	UF : 7, UT : 3,	CONFIG : 'F U T, 0, 0, 0',
	X =   -66.816  mm,	Y =   342.344  mm,	Z =     0.000  mm,
	W =  -167.363 deg,	P =     0.000 deg,	R =  -154.099 deg
};
P[1214]{
   GP1:
	UF : 7, UT : 3,	CONFIG : 'F U T, 0, 0, 0',
	X =   -66.816  mm,	Y =   342.344  mm,	Z =     0.000  mm,
	W =  -167.363 deg,	P =     0.000 deg,	R =  -154.099 deg
};
P[1215]{
   GP1:
	UF : 7, UT : 3,	CONFIG : 'F U T, 0, 0, 0',
	X =   -66.816  mm,	Y =   342.344  mm,	Z =     0.000  mm,
	W =  -167.363 deg,	P =     0.000 deg,	R =  -154.099 deg
};
P[1216]{
   GP1:
	UF : 7, UT : 3,	CONFIG : 'F U T, 0, 0, 0',
	X =   -46.005  mm,	Y =   345.765  mm,	Z =     0.000  mm,
	W =  -167.363 deg,	P =     0.000 deg,	R =  -157.374 deg
};
P[1217]{
   GP1:
	UF : 7, UT : 3,	CONFIG : 'F U T, 0, 0, 0',
	X =   -26.635  mm,	Y =   347.781  mm,	Z =     0.000  mm,
	W =  -167.364 deg,	P =     0.000 deg,	R =  -160.858 deg
};
P[1218]{
   GP1:
	UF : 7, UT : 3,	CONFIG : 'F U T, 0, 0, 0',
	X =   -26.635  mm,	Y =   347.781  mm,	Z =     0.000  mm,
	W =  -167.364 deg,	P =     0.000 deg,	R =  -160.858 deg
};
P[1219]{
   GP1:
	UF : 7, UT : 3,	CONFIG : 'F U T, 0, 0, 0',
	X =   -26.635  mm,	Y =   347.781  mm,	Z =     0.000  mm,
	W =  -167.364 deg,	P =     0.000 deg,	R =  -160.858 deg
};
P[1220]{
   GP1:
	UF : 7, UT : 3,	CONFIG : 'F U T, 0, 0, 0',
	X =   -26.635  mm,	Y =   347.781  mm,	Z =     0.000  mm,
	W =  -167.364 deg,	P =     0.000 deg,	R =  -160.858 deg
};
P[1221]{
   GP1:
	UF : 7, UT : 3,	CONFIG : 'F U T, 0, 0, 0',
	X =    26.635  mm,	Y =   347.781  mm,	Z =     0.000  mm,
	W =  -167.363 deg,	P =     0.000 deg,	R =  -169.046 deg
};
P[1222]{
   GP1:
	UF : 7, UT : 3,	CONFIG : 'F U T, 0, 0, 0',
	X =    26.635  mm,	Y =   347.781  mm,	Z =     0.000  mm,
	W =  -167.363 deg,	P =     0.000 deg,	R =  -169.046 deg
};
P[1223]{
   GP1:
	UF : 7, UT : 3,	CONFIG : 'F U T, 0, 0, 0',
	X =    26.635  mm,	Y =   347.781  mm,	Z =     0.000  mm,
	W =  -167.363 deg,	P =     0.000 deg,	R =  -169.046 deg
};
P[1224]{
   GP1:
	UF : 7, UT : 3,	CONFIG : 'F U T, 0, 0, 0',
	X =    26.635  mm,	Y =   347.781  mm,	Z =     0.000  mm,
	W =  -167.363 deg,	P =     0.000 deg,	R =  -169.046 deg
};
P[1225]{
   GP1:
	UF : 7, UT : 3,	CONFIG : 'F U T, 0, 0, 0',
	X =    45.934  mm,	Y =   345.776  mm,	Z =     0.000  mm,
	W =  -167.363 deg,	P =     0.000 deg,	R =  -172.500 deg
};
P[1226]{
   GP1:
	UF : 7, UT : 3,	CONFIG : 'F U T, 0, 0, 0',
	X =    66.816  mm,	Y =   342.344  mm,	Z =     0.000  mm,
	W =  -167.363 deg,	P =     0.000 deg,	R =  -175.771 deg
};
P[1227]{
   GP1:
	UF : 7, UT : 3,	CONFIG : 'F U T, 0, 0, 0',
	X =    66.816  mm,	Y =   342.344  mm,	Z =     0.000  mm,
	W =  -167.363 deg,	P =     0.000 deg,	R =  -175.771 deg
};
P[1228]{
   GP1:
	UF : 7, UT : 3,	CONFIG : 'F U T, 0, 0, 0',
	X =    66.816  mm,	Y =   342.344  mm,	Z =     0.000  mm,
	W =  -167.363 deg,	P =     0.000 deg,	R =  -175.771 deg
};
P[1229]{
   GP1:
	UF : 7, UT : 3,	CONFIG : 'F U T, 0, 0, 0',
	X =    66.816  mm,	Y =   342.344  mm,	Z =     0.000  mm,
	W =  -167.363 deg,	P =     0.000 deg,	R =  -175.771 deg
};
P[1230]{
   GP1:
	UF : 7, UT : 3,	CONFIG : 'F U T, 0, 0, 0',
	X =    88.319  mm,	Y =   337.433  mm,	Z =     0.000  mm,
	W =  -167.363 deg,	P =     0.000 deg,	R =  -179.012 deg
};
P[1231]{
   GP1:
	UF : 7, UT : 3,	CONFIG : 'F U T, 0, 0, 0',
	X =    88.319  mm,	Y =   337.433  mm,	Z =     0.000  mm,
	W =  -167.363 deg,	P =     0.000 deg,	R =  -179.012 deg
};
P[1232]{
   GP1:
	UF : 7, UT : 3,	CONFIG : 'F U T, 0, 0, 0',
	X =    88.319  mm,	Y =   337.433  mm,	Z =     0.000  mm,
	W =  -167.363 deg,	P =     0.000 deg,	R =  -179.012 deg
};
P[1233]{
   GP1:
	UF : 7, UT : 3,	CONFIG : 'F U T, 0, 0, 0',
	X =    88.319  mm,	Y =   337.433  mm,	Z =     0.000  mm,
	W =  -167.363 deg,	P =     0.000 deg,	R =  -179.012 deg
};
P[1234]{
   GP1:
	UF : 7, UT : 3,	CONFIG : 'F U T, 0, 0, 0',
	X =   106.083  mm,	Y =   332.287  mm,	Z =     0.000  mm,
	W =  -167.364 deg,	P =     0.000 deg,	R =   177.374 deg
};
P[1235]{
   GP1:
	UF : 7, UT : 3,	CONFIG : 'F U T, 0, 0, 0',
	X =   126.912  mm,	Y =   324.901  mm,	Z =     0.000  mm,
	W =  -167.364 deg,	P =     0.000 deg,	R =   174.134 deg
};
P[1236]{
   GP1:
	UF : 7, UT : 3,	CONFIG : 'F U T, 0, 0, 0',
	X =   126.912  mm,	Y =   324.901  mm,	Z =     0.000  mm,
	W =  -167.364 deg,	P =     0.000 deg,	R =   174.134 deg
};
P[1237]{
   GP1:
	UF : 7, UT : 3,	CONFIG : 'F U T, 0, 0, 0',
	X =   126.912  mm,	Y =   324.901  mm,	Z =     0.000  mm,
	W =  -167.364 deg,	P =     0.000 deg,	R =   174.134 deg
};
P[1238]{
   GP1:
	UF : 7, UT : 3,	CONFIG : 'F U T, 0, 0, 0',
	X =   126.912  mm,	Y =   324.901  mm,	Z =     0.000  mm,
	W =  -167.364 deg,	P =     0.000 deg,	R =   174.134 deg
};
P[1239]{
   GP1:
	UF : 7, UT : 3,	CONFIG : 'F U T, 0, 0, 0',
	X =   174.892  mm,	Y =   301.790  mm,	Z =     0.000  mm,
	W =  -167.364 deg,	P =     0.001 deg,	R =   165.335 deg
};
P[1240]{
   GP1:
	UF : 7, UT : 3,	CONFIG : 'F U T, 0, 0, 0',
	X =   174.892  mm,	Y =   301.790  mm,	Z =     0.000  mm,
	W =  -167.364 deg,	P =     0.001 deg,	R =   165.335 deg
};
P[1241]{
   GP1:
	UF : 7, UT : 3,	CONFIG : 'F U T, 0, 0, 0',
	X =   174.892  mm,	Y =   301.790  mm,	Z =     0.000  mm,
	W =  -167.364 deg,	P =     0.001 deg,	R =   165.335 deg
};
P[1242]{
   GP1:
	UF : 7, UT : 3,	CONFIG : 'F U T, 0, 0, 0',
	X =   174.892  mm,	Y =   301.790  mm,	Z =     0.000  mm,
	W =  -167.364 deg,	P =     0.001 deg,	R =   165.335 deg
};
P[1243]{
   GP1:
	UF : 7, UT : 3,	CONFIG : 'F U T, 0, 0, 0',
	X =   191.564  mm,	Y =   291.498  mm,	Z =     0.000  mm,
	W =  -167.364 deg,	P =     0.000 deg,	R =   161.703 deg
};
P[1244]{
   GP1:
	UF : 7, UT : 3,	CONFIG : 'F U T, 0, 0, 0',
	X =   208.616  mm,	Y =   279.549  mm,	Z =     0.000  mm,
	W =  -167.364 deg,	P =     0.000 deg,	R =   158.339 deg
};
P[1245]{
   GP1:
	UF : 7, UT : 3,	CONFIG : 'F U T, 0, 0, 0',
	X =   224.914  mm,	Y =   266.601  mm,	Z =     0.001  mm,
	W =  -167.364 deg,	P =     0.000 deg,	R =   154.951 deg
};
P[1246]{
   GP1:
	UF : 7, UT : 3,	CONFIG : 'F U T, 0, 0, 0',
	X =   239.976  mm,	Y =   253.131  mm,	Z =     0.000  mm,
	W =  -167.365 deg,	P =     0.000 deg,	R =   151.474 deg
};
P[1247]{
   GP1:
	UF : 7, UT : 3,	CONFIG : 'F U T, 0, 0, 0',
	X =   255.318  mm,	Y =   237.661  mm,	Z =     0.000  mm,
	W =  -167.365 deg,	P =    -0.001 deg,	R =   148.214 deg
};
P[1248]{
   GP1:
	UF : 7, UT : 3,	CONFIG : 'F U T, 0, 0, 0',
	X =   255.318  mm,	Y =   237.661  mm,	Z =     0.000  mm,
	W =  -167.365 deg,	P =    -0.001 deg,	R =   148.214 deg
};
P[1249]{
   GP1:
	UF : 7, UT : 3,	CONFIG : 'F U T, 0, 0, 0',
	X =   255.318  mm,	Y =   237.661  mm,	Z =     0.000  mm,
	W =  -167.365 deg,	P =    -0.001 deg,	R =   148.214 deg
};
P[1250]{
   GP1:
	UF : 7, UT : 3,	CONFIG : 'F U T, 0, 0, 0',
	X =   255.318  mm,	Y =   237.661  mm,	Z =     0.000  mm,
	W =  -167.365 deg,	P =    -0.001 deg,	R =   148.214 deg
};
P[1251]{
   GP1:
	UF : 7, UT : 3,	CONFIG : 'F U T, 0, 0, 0',
	X =   288.517  mm,	Y =   196.042  mm,	Z =     0.000  mm,
	W =  -167.364 deg,	P =     0.001 deg,	R =   138.644 deg
};
P[1252]{
   GP1:
	UF : 7, UT : 3,	CONFIG : 'F U T, 0, 0, 0',
	X =   288.517  mm,	Y =   196.042  mm,	Z =     0.000  mm,
	W =  -167.364 deg,	P =     0.001 deg,	R =   138.644 deg
};
P[1253]{
   GP1:
	UF : 7, UT : 3,	CONFIG : 'F U T, 0, 0, 0',
	X =   288.517  mm,	Y =   196.042  mm,	Z =     0.000  mm,
	W =  -167.364 deg,	P =     0.001 deg,	R =   138.644 deg
};
P[1254]{
   GP1:
	UF : 7, UT : 3,	CONFIG : 'F U T, 0, 0, 0',
	X =   288.517  mm,	Y =   196.042  mm,	Z =     0.000  mm,
	W =  -167.364 deg,	P =     0.001 deg,	R =   138.644 deg
};
P[1255]{
   GP1:
	UF : 7, UT : 3,	CONFIG : 'F U T, 0, 0, 0',
	X =   300.602  mm,	Y =   176.942  mm,	Z =     0.000  mm,
	W =  -167.364 deg,	P =     0.000 deg,	R =   135.546 deg
};
P[1256]{
   GP1:
	UF : 7, UT : 3,	CONFIG : 'F U T, 0, 0, 0',
	X =   309.321  mm,	Y =   161.197  mm,	Z =     0.000  mm,
	W =  -167.363 deg,	P =     0.000 deg,	R =   132.101 deg
};
P[1257]{
   GP1:
	UF : 7, UT : 3,	CONFIG : 'F U T, 0, 0, 0',
	X =   309.321  mm,	Y =   161.197  mm,	Z =     0.000  mm,
	W =  -167.363 deg,	P =     0.000 deg,	R =   132.101 deg
};
P[1258]{
   GP1:
	UF : 7, UT : 3,	CONFIG : 'F U T, 0, 0, 0',
	X =   309.321  mm,	Y =   161.197  mm,	Z =     0.000  mm,
	W =  -167.363 deg,	P =     0.000 deg,	R =   132.101 deg
};
P[1259]{
   GP1:
	UF : 7, UT : 3,	CONFIG : 'F U T, 0, 0, 0',
	X =   309.321  mm,	Y =   161.197  mm,	Z =     0.000  mm,
	W =  -167.363 deg,	P =     0.000 deg,	R =   132.101 deg
};
P[1260]{
   GP1:
	UF : 7, UT : 3,	CONFIG : 'F U T, 0, 0, 0',
	X =   318.900  mm,	Y =   141.321  mm,	Z =     0.000  mm,
	W =  -167.363 deg,	P =     0.000 deg,	R =   128.500 deg
};
P[1261]{
   GP1:
	UF : 7, UT : 3,	CONFIG : 'F U T, 0, 0, 0',
	X =   318.900  mm,	Y =   141.321  mm,	Z =     0.000  mm,
	W =  -167.363 deg,	P =     0.000 deg,	R =   128.500 deg
};
P[1262]{
   GP1:
	UF : 7, UT : 3,	CONFIG : 'F U T, 0, 0, 0',
	X =   318.900  mm,	Y =   141.321  mm,	Z =     0.000  mm,
	W =  -167.363 deg,	P =     0.000 deg,	R =   128.500 deg
};
P[1263]{
   GP1:
	UF : 7, UT : 3,	CONFIG : 'F U T, 0, 0, 0',
	X =   318.900  mm,	Y =   141.321  mm,	Z =     0.000  mm,
	W =  -167.363 deg,	P =     0.000 deg,	R =   128.500 deg
};
P[1264]{
   GP1:
	UF : 7, UT : 3,	CONFIG : 'F U T, 0, 0, 0',
	X =   327.247  mm,	Y =   120.740  mm,	Z =     0.000  mm,
	W =  -167.364 deg,	P =     0.000 deg,	R =   125.297 deg
};
P[1265]{
   GP1:
	UF : 7, UT : 3,	CONFIG : 'F U T, 0, 0, 0',
	X =   333.135  mm,	Y =   103.355  mm,	Z =     0.000  mm,
	W =  -167.365 deg,	P =    -0.001 deg,	R =   121.761 deg
};
P[1266]{
   GP1:
	UF : 7, UT : 3,	CONFIG : 'F U T, 0, 0, 0',
	X =   333.135  mm,	Y =   103.355  mm,	Z =     0.000  mm,
	W =  -167.365 deg,	P =    -0.001 deg,	R =   121.761 deg
};
P[1267]{
   GP1:
	UF : 7, UT : 3,	CONFIG : 'F U T, 0, 0, 0',
	X =   333.135  mm,	Y =   103.355  mm,	Z =     0.000  mm,
	W =  -167.365 deg,	P =    -0.001 deg,	R =   121.761 deg
};
P[1268]{
   GP1:
	UF : 7, UT : 3,	CONFIG : 'F U T, 0, 0, 0',
	X =   333.135  mm,	Y =   103.355  mm,	Z =     0.000  mm,
	W =  -167.365 deg,	P =    -0.001 deg,	R =   121.761 deg
};
P[1269]{
   GP1:
	UF : 7, UT : 3,	CONFIG : 'F U T, 0, 0, 0',
	X =   344.991  mm,	Y =    51.425  mm,	Z =     0.000  mm,
	W =  -167.364 deg,	P =     0.001 deg,	R =   113.386 deg
};
P[1270]{
   GP1:
	UF : 7, UT : 3,	CONFIG : 'F U T, 0, 0, 0',
	X =   344.991  mm,	Y =    51.425  mm,	Z =     0.000  mm,
	W =  -167.364 deg,	P =     0.001 deg,	R =   113.386 deg
};
P[1271]{
   GP1:
	UF : 7, UT : 3,	CONFIG : 'F U T, 0, 0, 0',
	X =   344.991  mm,	Y =    51.425  mm,	Z =     0.000  mm,
	W =  -167.364 deg,	P =     0.001 deg,	R =   113.386 deg
};
P[1272]{
   GP1:
	UF : 7, UT : 3,	CONFIG : 'F U T, 0, 0, 0',
	X =   344.991  mm,	Y =    51.425  mm,	Z =     0.000  mm,
	W =  -167.364 deg,	P =     0.001 deg,	R =   113.386 deg
};
P[1273]{
   GP1:
	UF : 7, UT : 3,	CONFIG : 'F U T, 0, 0, 0',
	X =   347.736  mm,	Y =    27.239  mm,	Z =     0.000  mm,
	W =  -167.364 deg,	P =     0.000 deg,	R =   109.541 deg
};
P[1274]{
   GP1:
	UF : 7, UT : 3,	CONFIG : 'F U T, 0, 0, 0',
	X =   348.821  mm,	Y =     0.000  mm,	Z =     0.000  mm,
	W =  -167.364 deg,	P =    -0.001 deg,	R =   105.687 deg
};
P[1275]{
   GP1:
	UF : 7, UT : 3,	CONFIG : 'F U T, 0, 0, 0',
	X =   348.821  mm,	Y =     0.000  mm,	Z =     0.000  mm,
	W =  -167.364 deg,	P =    -0.001 deg,	R =   105.687 deg
};
P[1276]{
   GP1:
	UF : 7, UT : 3,	CONFIG : 'F U T, 0, 0, 0',
	X =   348.821  mm,	Y =     0.000  mm,	Z =     0.000  mm,
	W =  -167.364 deg,	P =    -0.001 deg,	R =   105.687 deg
};
P[1277]{
   GP1:
	UF : 7, UT : 3,	CONFIG : 'F U T, 0, 0, 0',
	X =   348.821  mm,	Y =     0.000  mm,	Z =     0.000  mm,
	W =  -167.364 deg,	P =    -0.001 deg,	R =   105.687 deg
};
P[1278]{
   GP1:
	UF : 7, UT : 3,	CONFIG : 'F U T, 0, 0, 0',
	X =   345.686  mm,	Y =     0.000  mm,	Z =     0.000  mm,
	W =  -167.364 deg,	P =    -0.001 deg,	R =   105.687 deg
};
P[1279]{
   GP1:
	UF : 7, UT : 3,	CONFIG : 'F U T, 0, 0, 0',
	X =   345.686  mm,	Y =     0.000  mm,	Z =     0.000  mm,
	W =  -167.364 deg,	P =    -0.001 deg,	R =   105.687 deg
};
P[1280]{
   GP1:
	UF : 7, UT : 3,	CONFIG : 'F U T, 0, 0, 0',
	X =   345.686  mm,	Y =     0.000  mm,	Z =     0.000  mm,
	W =  -167.364 deg,	P =    -0.001 deg,	R =   105.687 deg
};
P[1281]{
   GP1:
	UF : 7, UT : 3,	CONFIG : 'F U T, 0, 0, 0',
	X =   345.686  mm,	Y =     0.000  mm,	Z =     0.000  mm,
	W =  -167.364 deg,	P =    -0.001 deg,	R =   105.687 deg
};
P[1282]{
   GP1:
	UF : 7, UT : 3,	CONFIG : 'F U T, 0, 0, 0',
	X =   344.660  mm,	Y =    26.365  mm,	Z =     0.000  mm,
	W =  -167.364 deg,	P =     0.000 deg,	R =   109.418 deg
};
P[1283]{
   GP1:
	UF : 7, UT : 3,	CONFIG : 'F U T, 0, 0, 0',
	X =   342.332  mm,	Y =    47.913  mm,	Z =     0.000  mm,
	W =  -167.364 deg,	P =     0.001 deg,	R =   113.455 deg
};
P[1284]{
   GP1:
	UF : 7, UT : 3,	CONFIG : 'F U T, 0, 0, 0',
	X =   342.332  mm,	Y =    47.913  mm,	Z =     0.000  mm,
	W =  -167.364 deg,	P =     0.001 deg,	R =   113.455 deg
};
P[1285]{
   GP1:
	UF : 7, UT : 3,	CONFIG : 'F U T, 0, 0, 0',
	X =   342.332  mm,	Y =    47.913  mm,	Z =     0.000  mm,
	W =  -167.364 deg,	P =     0.001 deg,	R =   113.455 deg
};
P[1286]{
   GP1:
	UF : 7, UT : 3,	CONFIG : 'F U T, 0, 0, 0',
	X =   342.332  mm,	Y =    47.913  mm,	Z =     0.000  mm,
	W =  -167.364 deg,	P =     0.001 deg,	R =   113.455 deg
};
P[1287]{
   GP1:
	UF : 7, UT : 3,	CONFIG : 'F U T, 0, 0, 0',
	X =   329.241  mm,	Y =   105.355  mm,	Z =     0.000  mm,
	W =  -167.365 deg,	P =    -0.001 deg,	R =   123.426 deg
};
P[1288]{
   GP1:
	UF : 7, UT : 3,	CONFIG : 'F U T, 0, 0, 0',
	X =   329.241  mm,	Y =   105.355  mm,	Z =     0.000  mm,
	W =  -167.365 deg,	P =    -0.001 deg,	R =   123.426 deg
};
P[1289]{
   GP1:
	UF : 7, UT : 3,	CONFIG : 'F U T, 0, 0, 0',
	X =   329.241  mm,	Y =   105.355  mm,	Z =     0.000  mm,
	W =  -167.365 deg,	P =    -0.001 deg,	R =   123.426 deg
};
P[1290]{
   GP1:
	UF : 7, UT : 3,	CONFIG : 'F U T, 0, 0, 0',
	X =   329.241  mm,	Y =   105.355  mm,	Z =     0.000  mm,
	W =  -167.365 deg,	P =    -0.001 deg,	R =   123.426 deg
};
P[1291]{
   GP1:
	UF : 7, UT : 3,	CONFIG : 'F U T, 0, 0, 0',
	X =   321.435  mm,	Y =   127.175  mm,	Z =     0.000  mm,
	W =  -167.364 deg,	P =     0.000 deg,	R =   126.652 deg
};
P[1292]{
   GP1:
	UF : 7, UT : 3,	CONFIG : 'F U T, 0, 0, 0',
	X =   314.243  mm,	Y =   144.001  mm,	Z =     0.000  mm,
	W =  -167.363 deg,	P =     0.000 deg,	R =   130.454 deg
};
P[1293]{
   GP1:
	UF : 7, UT : 3,	CONFIG : 'F U T, 0, 0, 0',
	X =   314.243  mm,	Y =   144.001  mm,	Z =     0.000  mm,
	W =  -167.363 deg,	P =     0.000 deg,	R =   130.454 deg
};
P[1294]{
   GP1:
	UF : 7, UT : 3,	CONFIG : 'F U T, 0, 0, 0',
	X =   314.243  mm,	Y =   144.001  mm,	Z =     0.000  mm,
	W =  -167.363 deg,	P =     0.000 deg,	R =   130.454 deg
};
P[1295]{
   GP1:
	UF : 7, UT : 3,	CONFIG : 'F U T, 0, 0, 0',
	X =   314.243  mm,	Y =   144.001  mm,	Z =     0.000  mm,
	W =  -167.363 deg,	P =     0.000 deg,	R =   130.454 deg
};
P[1296]{
   GP1:
	UF : 7, UT : 3,	CONFIG : 'F U T, 0, 0, 0',
	X =   308.505  mm,	Y =   155.937  mm,	Z =     0.000  mm,
	W =  -167.363 deg,	P =     0.000 deg,	R =   132.305 deg
};
P[1297]{
   GP1:
	UF : 7, UT : 3,	CONFIG : 'F U T, 0, 0, 0',
	X =   308.505  mm,	Y =   155.937  mm,	Z =     0.000  mm,
	W =  -167.363 deg,	P =     0.000 deg,	R =   132.305 deg
};
P[1298]{
   GP1:
	UF : 7, UT : 3,	CONFIG : 'F U T, 0, 0, 0',
	X =   308.505  mm,	Y =   155.937  mm,	Z =     0.000  mm,
	W =  -167.363 deg,	P =     0.000 deg,	R =   132.305 deg
};
P[1299]{
   GP1:
	UF : 7, UT : 3,	CONFIG : 'F U T, 0, 0, 0',
	X =   308.505  mm,	Y =   155.937  mm,	Z =     0.000  mm,
	W =  -167.363 deg,	P =     0.000 deg,	R =   132.305 deg
};
P[1300]{
   GP1:
	UF : 7, UT : 3,	CONFIG : 'F U T, 0, 0, 0',
	X =   297.848  mm,	Y =   175.435  mm,	Z =     0.000  mm,
	W =  -167.364 deg,	P =     0.000 deg,	R =   135.574 deg
};
P[1301]{
   GP1:
	UF : 7, UT : 3,	CONFIG : 'F U T, 0, 0, 0',
	X =   287.641  mm,	Y =   191.697  mm,	Z =     0.000  mm,
	W =  -167.364 deg,	P =     0.001 deg,	R =   138.948 deg
};
P[1302]{
   GP1:
	UF : 7, UT : 3,	CONFIG : 'F U T, 0, 0, 0',
	X =   287.641  mm,	Y =   191.697  mm,	Z =     0.000  mm,
	W =  -167.364 deg,	P =     0.001 deg,	R =   138.948 deg
};
P[1303]{
   GP1:
	UF : 7, UT : 3,	CONFIG : 'F U T, 0, 0, 0',
	X =   287.641  mm,	Y =   191.697  mm,	Z =     0.000  mm,
	W =  -167.364 deg,	P =     0.001 deg,	R =   138.948 deg
};
P[1304]{
   GP1:
	UF : 7, UT : 3,	CONFIG : 'F U T, 0, 0, 0',
	X =   287.641  mm,	Y =   191.697  mm,	Z =     0.000  mm,
	W =  -167.364 deg,	P =     0.001 deg,	R =   138.948 deg
};
P[1305]{
   GP1:
	UF : 7, UT : 3,	CONFIG : 'F U T, 0, 0, 0',
	X =   250.901  mm,	Y =   237.773  mm,	Z =     0.000  mm,
	W =  -167.365 deg,	P =    -0.001 deg,	R =   148.657 deg
};
P[1306]{
   GP1:
	UF : 7, UT : 3,	CONFIG : 'F U T, 0, 0, 0',
	X =   250.901  mm,	Y =   237.773  mm,	Z =     0.000  mm,
	W =  -167.365 deg,	P =    -0.001 deg,	R =   148.657 deg
};
P[1307]{
   GP1:
	UF : 7, UT : 3,	CONFIG : 'F U T, 0, 0, 0',
	X =   250.901  mm,	Y =   237.773  mm,	Z =     0.000  mm,
	W =  -167.365 deg,	P =    -0.001 deg,	R =   148.657 deg
};
P[1308]{
   GP1:
	UF : 7, UT : 3,	CONFIG : 'F U T, 0, 0, 0',
	X =   250.901  mm,	Y =   237.773  mm,	Z =     0.000  mm,
	W =  -167.365 deg,	P =    -0.001 deg,	R =   148.657 deg
};
P[1309]{
   GP1:
	UF : 7, UT : 3,	CONFIG : 'F U T, 0, 0, 0',
	X =   233.996  mm,	Y =   254.423  mm,	Z =     0.000  mm,
	W =  -167.365 deg,	P =     0.000 deg,	R =   152.488 deg
};
P[1310]{
   GP1:
	UF : 7, UT : 3,	CONFIG : 'F U T, 0, 0, 0',
	X =   216.033  mm,	Y =   269.842  mm,	Z =     0.001  mm,
	W =  -167.364 deg,	P =     0.000 deg,	R =   156.343 deg
};
P[1311]{
   GP1:
	UF : 7, UT : 3,	CONFIG : 'F U T, 0, 0, 0',
	X =   197.478  mm,	Y =   283.704  mm,	Z =     0.000  mm,
	W =  -167.364 deg,	P =     0.000 deg,	R =   160.254 deg
};
P[1312]{
   GP1:
	UF : 7, UT : 3,	CONFIG : 'F U T, 0, 0, 0',
	X =   175.979  mm,	Y =   297.529  mm,	Z =     0.000  mm,
	W =  -167.364 deg,	P =     0.001 deg,	R =   164.017 deg
};
P[1313]{
   GP1:
	UF : 7, UT : 3,	CONFIG : 'F U T, 0, 0, 0',
	X =   175.979  mm,	Y =   297.529  mm,	Z =     0.000  mm,
	W =  -167.364 deg,	P =     0.001 deg,	R =   164.017 deg
};
P[1314]{
   GP1:
	UF : 7, UT : 3,	CONFIG : 'F U T, 0, 0, 0',
	X =   175.979  mm,	Y =   297.529  mm,	Z =     0.000  mm,
	W =  -167.364 deg,	P =     0.001 deg,	R =   164.017 deg
};
P[1315]{
   GP1:
	UF : 7, UT : 3,	CONFIG : 'F U T, 0, 0, 0',
	X =   175.979  mm,	Y =   297.529  mm,	Z =     0.000  mm,
	W =  -167.364 deg,	P =     0.001 deg,	R =   164.017 deg
};
P[1316]{
   GP1:
	UF : 7, UT : 3,	CONFIG : 'F U T, 0, 0, 0',
	X =   122.884  mm,	Y =   323.086  mm,	Z =     0.000  mm,
	W =  -167.364 deg,	P =     0.000 deg,	R =   173.711 deg
};
P[1317]{
   GP1:
	UF : 7, UT : 3,	CONFIG : 'F U T, 0, 0, 0',
	X =   122.884  mm,	Y =   323.086  mm,	Z =     0.000  mm,
	W =  -167.364 deg,	P =     0.000 deg,	R =   173.711 deg
};
P[1318]{
   GP1:
	UF : 7, UT : 3,	CONFIG : 'F U T, 0, 0, 0',
	X =   122.884  mm,	Y =   323.086  mm,	Z =     0.000  mm,
	W =  -167.364 deg,	P =     0.000 deg,	R =   173.711 deg
};
P[1319]{
   GP1:
	UF : 7, UT : 3,	CONFIG : 'F U T, 0, 0, 0',
	X =   122.884  mm,	Y =   323.086  mm,	Z =     0.000  mm,
	W =  -167.364 deg,	P =     0.000 deg,	R =   173.711 deg
};
P[1320]{
   GP1:
	UF : 7, UT : 3,	CONFIG : 'F U T, 0, 0, 0',
	X =   105.120  mm,	Y =   329.306  mm,	Z =     0.000  mm,
	W =  -167.364 deg,	P =     0.000 deg,	R =   177.352 deg
};
P[1321]{
   GP1:
	UF : 7, UT : 3,	CONFIG : 'F U T, 0, 0, 0',
	X =    83.393  mm,	Y =   335.476  mm,	Z =     0.000  mm,
	W =  -167.363 deg,	P =     0.000 deg,	R =  -179.548 deg
};
P[1322]{
   GP1:
	UF : 7, UT : 3,	CONFIG : 'F U T, 0, 0, 0',
	X =    83.393  mm,	Y =   335.476  mm,	Z =     0.000  mm,
	W =  -167.363 deg,	P =     0.000 deg,	R =  -179.548 deg
};
P[1323]{
   GP1:
	UF : 7, UT : 3,	CONFIG : 'F U T, 0, 0, 0',
	X =    83.393  mm,	Y =   335.476  mm,	Z =     0.000  mm,
	W =  -167.363 deg,	P =     0.000 deg,	R =  -179.548 deg
};
P[1324]{
   GP1:
	UF : 7, UT : 3,	CONFIG : 'F U T, 0, 0, 0',
	X =    83.393  mm,	Y =   335.476  mm,	Z =     0.000  mm,
	W =  -167.363 deg,	P =     0.000 deg,	R =  -179.548 deg
};
P[1325]{
   GP1:
	UF : 7, UT : 3,	CONFIG : 'F U T, 0, 0, 0',
	X =    70.462  mm,	Y =   338.412  mm,	Z =     0.000  mm,
	W =  -167.363 deg,	P =     0.000 deg,	R =  -177.098 deg
};
P[1326]{
   GP1:
	UF : 7, UT : 3,	CONFIG : 'F U T, 0, 0, 0',
	X =    70.462  mm,	Y =   338.412  mm,	Z =     0.000  mm,
	W =  -167.363 deg,	P =     0.000 deg,	R =  -177.098 deg
};
P[1327]{
   GP1:
	UF : 7, UT : 3,	CONFIG : 'F U T, 0, 0, 0',
	X =    70.462  mm,	Y =   338.412  mm,	Z =     0.000  mm,
	W =  -167.363 deg,	P =     0.000 deg,	R =  -177.098 deg
};
P[1328]{
   GP1:
	UF : 7, UT : 3,	CONFIG : 'F U T, 0, 0, 0',
	X =    70.462  mm,	Y =   338.412  mm,	Z =     0.000  mm,
	W =  -167.363 deg,	P =     0.000 deg,	R =  -177.098 deg
};
P[1329]{
   GP1:
	UF : 7, UT : 3,	CONFIG : 'F U T, 0, 0, 0',
	X =    51.004  mm,	Y =   341.888  mm,	Z =     0.000  mm,
	W =  -167.363 deg,	P =     0.000 deg,	R =  -173.340 deg
};
P[1330]{
   GP1:
	UF : 7, UT : 3,	CONFIG : 'F U T, 0, 0, 0',
	X =    29.459  mm,	Y =   344.419  mm,	Z =     0.000  mm,
	W =  -167.363 deg,	P =     0.000 deg,	R =  -169.941 deg
};
P[1331]{
   GP1:
	UF : 7, UT : 3,	CONFIG : 'F U T, 0, 0, 0',
	X =    29.459  mm,	Y =   344.419  mm,	Z =     0.000  mm,
	W =  -167.363 deg,	P =     0.000 deg,	R =  -169.941 deg
};
P[1332]{
   GP1:
	UF : 7, UT : 3,	CONFIG : 'F U T, 0, 0, 0',
	X =    29.459  mm,	Y =   344.419  mm,	Z =     0.000  mm,
	W =  -167.363 deg,	P =     0.000 deg,	R =  -169.941 deg
};
P[1333]{
   GP1:
	UF : 7, UT : 3,	CONFIG : 'F U T, 0, 0, 0',
	X =    29.459  mm,	Y =   344.419  mm,	Z =     0.000  mm,
	W =  -167.363 deg,	P =     0.000 deg,	R =  -169.941 deg
};
P[1334]{
   GP1:
	UF : 7, UT : 3,	CONFIG : 'F U T, 0, 0, 0',
	X =   -29.459  mm,	Y =   344.419  mm,	Z =     0.000  mm,
	W =  -167.364 deg,	P =     0.000 deg,	R =  -159.946 deg
};
P[1335]{
   GP1:
	UF : 7, UT : 3,	CONFIG : 'F U T, 0, 0, 0',
	X =   -29.459  mm,	Y =   344.419  mm,	Z =     0.000  mm,
	W =  -167.364 deg,	P =     0.000 deg,	R =  -159.946 deg
};
P[1336]{
   GP1:
	UF : 7, UT : 3,	CONFIG : 'F U T, 0, 0, 0',
	X =   -29.459  mm,	Y =   344.419  mm,	Z =     0.000  mm,
	W =  -167.364 deg,	P =     0.000 deg,	R =  -159.946 deg
};
P[1337]{
   GP1:
	UF : 7, UT : 3,	CONFIG : 'F U T, 0, 0, 0',
	X =   -29.459  mm,	Y =   344.419  mm,	Z =     0.000  mm,
	W =  -167.364 deg,	P =     0.000 deg,	R =  -159.946 deg
};
P[1338]{
   GP1:
	UF : 7, UT : 3,	CONFIG : 'F U T, 0, 0, 0',
	X =   -50.881  mm,	Y =   341.905  mm,	Z =     0.000  mm,
	W =  -167.363 deg,	P =     0.000 deg,	R =  -156.562 deg
};
P[1339]{
   GP1:
	UF : 7, UT : 3,	CONFIG : 'F U T, 0, 0, 0',
	X =   -70.462  mm,	Y =   338.412  mm,	Z =     0.000  mm,
	W =  -167.363 deg,	P =     0.000 deg,	R =  -152.846 deg
};
P[1340]{
   GP1:
	UF : 7, UT : 3,	CONFIG : 'F U T, 0, 0, 0',
	X =   -70.462  mm,	Y =   338.412  mm,	Z =     0.000  mm,
	W =  -167.363 deg,	P =     0.000 deg,	R =  -152.846 deg
};
P[1341]{
   GP1:
	UF : 7, UT : 3,	CONFIG : 'F U T, 0, 0, 0',
	X =   -70.462  mm,	Y =   338.412  mm,	Z =     0.000  mm,
	W =  -167.363 deg,	P =     0.000 deg,	R =  -152.846 deg
};
P[1342]{
   GP1:
	UF : 7, UT : 3,	CONFIG : 'F U T, 0, 0, 0',
	X =   -70.462  mm,	Y =   338.412  mm,	Z =     0.000  mm,
	W =  -167.363 deg,	P =     0.000 deg,	R =  -152.846 deg
};
P[1343]{
   GP1:
	UF : 7, UT : 3,	CONFIG : 'F U T, 0, 0, 0',
	X =   -83.393  mm,	Y =   335.476  mm,	Z =     0.000  mm,
	W =  -167.363 deg,	P =     0.000 deg,	R =  -150.369 deg
};
P[1344]{
   GP1:
	UF : 7, UT : 3,	CONFIG : 'F U T, 0, 0, 0',
	X =   -83.393  mm,	Y =   335.476  mm,	Z =     0.000  mm,
	W =  -167.363 deg,	P =     0.000 deg,	R =  -150.369 deg
};
P[1345]{
   GP1:
	UF : 7, UT : 3,	CONFIG : 'F U T, 0, 0, 0',
	X =   -83.393  mm,	Y =   335.476  mm,	Z =     0.000  mm,
	W =  -167.363 deg,	P =     0.000 deg,	R =  -150.369 deg
};
P[1346]{
   GP1:
	UF : 7, UT : 3,	CONFIG : 'F U T, 0, 0, 0',
	X =   -83.393  mm,	Y =   335.476  mm,	Z =     0.000  mm,
	W =  -167.363 deg,	P =     0.000 deg,	R =  -150.369 deg
};
P[1347]{
   GP1:
	UF : 7, UT : 3,	CONFIG : 'F U T, 0, 0, 0',
	X =  -105.618  mm,	Y =   329.150  mm,	Z =     0.000  mm,
	W =  -167.364 deg,	P =     0.001 deg,	R =  -147.148 deg
};
P[1348]{
   GP1:
	UF : 7, UT : 3,	CONFIG : 'F U T, 0, 0, 0',
	X =  -122.884  mm,	Y =   323.086  mm,	Z =     0.000  mm,
	W =  -167.364 deg,	P =     0.002 deg,	R =  -143.543 deg
};
P[1349]{
   GP1:
	UF : 7, UT : 3,	CONFIG : 'F U T, 0, 0, 0',
	X =  -122.884  mm,	Y =   323.086  mm,	Z =     0.000  mm,
	W =  -167.364 deg,	P =     0.002 deg,	R =  -143.543 deg
};
P[1350]{
   GP1:
	UF : 7, UT : 3,	CONFIG : 'F U T, 0, 0, 0',
	X =  -122.884  mm,	Y =   323.086  mm,	Z =     0.000  mm,
	W =  -167.364 deg,	P =     0.002 deg,	R =  -143.543 deg
};
P[1351]{
   GP1:
	UF : 7, UT : 3,	CONFIG : 'F U T, 0, 0, 0',
	X =  -122.884  mm,	Y =   323.086  mm,	Z =     0.000  mm,
	W =  -167.364 deg,	P =     0.002 deg,	R =  -143.543 deg
};
P[1352]{
   GP1:
	UF : 7, UT : 3,	CONFIG : 'F U T, 0, 0, 0',
	X =  -175.979  mm,	Y =   297.529  mm,	Z =     0.000  mm,
	W =  -167.373 deg,	P =    -0.006 deg,	R =  -133.905 deg
};
P[1353]{
   GP1:
	UF : 7, UT : 3,	CONFIG : 'F U T, 0, 0, 0',
	X =  -175.979  mm,	Y =   297.529  mm,	Z =     0.000  mm,
	W =  -167.373 deg,	P =    -0.006 deg,	R =  -133.905 deg
};
P[1354]{
   GP1:
	UF : 7, UT : 3,	CONFIG : 'F U T, 0, 0, 0',
	X =  -175.979  mm,	Y =   297.529  mm,	Z =     0.000  mm,
	W =  -167.373 deg,	P =    -0.006 deg,	R =  -133.905 deg
};
P[1355]{
   GP1:
	UF : 7, UT : 3,	CONFIG : 'F U T, 0, 0, 0',
	X =  -175.979  mm,	Y =   297.529  mm,	Z =     0.000  mm,
	W =  -167.373 deg,	P =    -0.006 deg,	R =  -133.905 deg
};
P[1356]{
   GP1:
	UF : 7, UT : 3,	CONFIG : 'F U T, 0, 0, 0',
	X =  -195.500  mm,	Y =   285.077  mm,	Z =     0.006  mm,
	W =  -167.372 deg,	P =    -0.005 deg,	R =  -130.444 deg
};
P[1357]{
   GP1:
	UF : 7, UT : 3,	CONFIG : 'F U T, 0, 0, 0',
	X =  -212.838  mm,	Y =   272.387  mm,	Z =     0.014  mm,
	W =  -167.372 deg,	P =    -0.004 deg,	R =  -126.946 deg
};
P[1358]{
   GP1:
	UF : 7, UT : 3,	CONFIG : 'F U T, 0, 0, 0',
	X =  -229.364  mm,	Y =   258.615  mm,	Z =     0.020  mm,
	W =  -167.371 deg,	P =    -0.003 deg,	R =  -123.454 deg
};
P[1359]{
   GP1:
	UF : 7, UT : 3,	CONFIG : 'F U T, 0, 0, 0',
	X =  -240.307  mm,	Y =   248.477  mm,	Z =     0.016  mm,
	W =  -167.396 deg,	P =     0.051 deg,	R =  -120.994 deg
};
P[1360]{
   GP1:
	UF : 7, UT : 3,	CONFIG : 'F U T, 0, 0, 0',
	X =  -250.901  mm,	Y =   237.773  mm,	Z =     0.000  mm,
	W =  -167.417 deg,	P =     0.107 deg,	R =  -118.546 deg
};
P[1361]{
   GP1:
	UF : 7, UT : 3,	CONFIG : 'F U T, 0, 0, 0',
	X =  -250.901  mm,	Y =   237.773  mm,	Z =     0.000  mm,
	W =  -167.417 deg,	P =     0.107 deg,	R =  -118.546 deg
};
P[1362]{
   GP1:
	UF : 7, UT : 3,	CONFIG : 'F U T, 0, 0, 0',
	X =  -250.901  mm,	Y =   237.773  mm,	Z =     0.000  mm,
	W =  -167.417 deg,	P =     0.107 deg,	R =  -118.546 deg
};
P[1363]{
   GP1:
	UF : 7, UT : 3,	CONFIG : 'F U T, 0, 0, 0',
	X =  -250.901  mm,	Y =   237.773  mm,	Z =     0.000  mm,
	W =  -167.417 deg,	P =     0.107 deg,	R =  -118.546 deg
};
P[1364]{
   GP1:
	UF : 7, UT : 3,	CONFIG : 'F U T, 0, 0, 0',
	X =  -287.641  mm,	Y =   191.697  mm,	Z =     0.000  mm,
	W =  -168.063 deg,	P =    -0.468 deg,	R =  -108.824 deg
};
P[1365]{
   GP1:
	UF : 7, UT : 3,	CONFIG : 'F U T, 0, 0, 0',
	X =  -287.641  mm,	Y =   191.697  mm,	Z =     0.000  mm,
	W =  -168.063 deg,	P =    -0.468 deg,	R =  -108.824 deg
};
P[1366]{
   GP1:
	UF : 7, UT : 3,	CONFIG : 'F U T, 0, 0, 0',
	X =  -287.641  mm,	Y =   191.697  mm,	Z =     0.000  mm,
	W =  -168.063 deg,	P =    -0.468 deg,	R =  -108.824 deg
};
P[1367]{
   GP1:
	UF : 7, UT : 3,	CONFIG : 'F U T, 0, 0, 0',
	X =  -287.641  mm,	Y =   191.697  mm,	Z =     0.000  mm,
	W =  -168.063 deg,	P =    -0.468 deg,	R =  -108.824 deg
};
P[1368]{
   GP1:
	UF : 7, UT : 3,	CONFIG : 'F U T, 0, 0, 0',
	X =  -295.473  mm,	Y =   179.397  mm,	Z =     0.299  mm,
	W =  -168.371 deg,	P =    -1.524 deg,	R =  -106.124 deg
};
P[1369]{
   GP1:
	UF : 7, UT : 3,	CONFIG : 'F U T, 0, 0, 0',
	X =  -299.979  mm,	Y =   171.757  mm,	Z =     0.593  mm,
	W =  -168.582 deg,	P =    -1.678 deg,	R =  -104.715 deg
};
P[1370]{
   GP1:
	UF : 7, UT : 3,	CONFIG : 'F U T, 0, 0, 0',
	X =  -304.573  mm,	Y =   163.495  mm,	Z =     0.880  mm,
	W =  -168.711 deg,	P =    -1.083 deg,	R =  -103.238 deg
};
P[1371]{
   GP1:
	UF : 7, UT : 3,	CONFIG : 'F U T, 0, 0, 0',
	X =  -307.581  mm,	Y =   157.753  mm,	Z =     1.000  mm,
	W =  -168.635 deg,	P =    -0.392 deg,	R =  -101.948 deg
};
P[1372]{
   GP1:
	UF : 7, UT : 3,	CONFIG : 'F U T, 0, 0, 0',
	X =  -307.581  mm,	Y =   157.753  mm,	Z =     1.000  mm,
	W =  -168.635 deg,	P =    -0.392 deg,	R =  -101.948 deg
};
P[1373]{
   GP1:
	UF : 7, UT : 3,	CONFIG : 'F U T, 0, 0, 0',
	X =  -307.581  mm,	Y =   157.753  mm,	Z =     1.000  mm,
	W =  -168.635 deg,	P =    -0.392 deg,	R =  -101.948 deg
};
P[1374]{
   GP1:
	UF : 7, UT : 3,	CONFIG : 'F U T, 0, 0, 0',
	X =  -307.581  mm,	Y =   157.753  mm,	Z =     1.000  mm,
	W =  -168.635 deg,	P =    -0.392 deg,	R =  -101.948 deg
};
P[1375]{
   GP1:
	UF : 7, UT : 3,	CONFIG : 'F U T, 0, 0, 0',
	X =  -315.125  mm,	Y =   142.110  mm,	Z =     1.000  mm,
	W =  -168.019 deg,	P =     0.716 deg,	R =   -99.203 deg
};
P[1376]{
   GP1:
	UF : 7, UT : 3,	CONFIG : 'F U T, 0, 0, 0',
	X =  -315.125  mm,	Y =   142.110  mm,	Z =     1.000  mm,
	W =  -168.019 deg,	P =     0.716 deg,	R =   -99.203 deg
};
P[1377]{
   GP1:
	UF : 7, UT : 3,	CONFIG : 'F U T, 0, 0, 0',
	X =  -315.125  mm,	Y =   142.110  mm,	Z =     1.000  mm,
	W =  -168.019 deg,	P =     0.716 deg,	R =   -99.203 deg
};
P[1378]{
   GP1:
	UF : 7, UT : 3,	CONFIG : 'F U T, 0, 0, 0',
	X =  -315.125  mm,	Y =   142.110  mm,	Z =     1.000  mm,
	W =  -168.019 deg,	P =     0.716 deg,	R =   -99.203 deg
};
P[1379]{
   GP1:
	UF : 7, UT : 3,	CONFIG : 'F U T, 0, 0, 0',
	X =  -319.199  mm,	Y =   132.690  mm,	Z =     0.839  mm,
	W =  -167.800 deg,	P =     1.582 deg,	R =   -97.400 deg
};
P[1380]{
   GP1:
	UF : 7, UT : 3,	CONFIG : 'F U T, 0, 0, 0',
	X =  -322.114  mm,	Y =   125.444  mm,	Z =     0.586  mm,
	W =  -167.715 deg,	P =     2.330 deg,	R =   -96.138 deg
};
P[1381]{
   GP1:
	UF : 7, UT : 3,	CONFIG : 'F U T, 0, 0, 0',
	X =  -324.359  mm,	Y =   119.513  mm,	Z =     0.341  mm,
	W =  -167.697 deg,	P =     2.244 deg,	R =   -95.130 deg
};
P[1382]{
   GP1:
	UF : 7, UT : 3,	CONFIG : 'F U T, 0, 0, 0',
	X =  -329.241  mm,	Y =   105.355  mm,	Z =     0.000  mm,
	W =  -167.650 deg,	P =     0.556 deg,	R =   -93.318 deg
};
P[1383]{
   GP1:
	UF : 7, UT : 3,	CONFIG : 'F U T, 0, 0, 0',
	X =  -329.241  mm,	Y =   105.355  mm,	Z =     0.000  mm,
	W =  -167.650 deg,	P =     0.556 deg,	R =   -93.318 deg
};
P[1384]{
   GP1:
	UF : 7, UT : 3,	CONFIG : 'F U T, 0, 0, 0',
	X =  -329.241  mm,	Y =   105.355  mm,	Z =     0.000  mm,
	W =  -167.650 deg,	P =     0.556 deg,	R =   -93.318 deg
};
P[1385]{
   GP1:
	UF : 7, UT : 3,	CONFIG : 'F U T, 0, 0, 0',
	X =  -329.241  mm,	Y =   105.355  mm,	Z =     0.000  mm,
	W =  -167.650 deg,	P =     0.556 deg,	R =   -93.318 deg
};
P[1386]{
   GP1:
	UF : 7, UT : 3,	CONFIG : 'F U T, 0, 1, 0',
	X =  -342.332  mm,	Y =    47.913  mm,	Z =     0.000  mm,
	W =  -167.380 deg,	P =    -0.011 deg,	R =   -83.337 deg
};
P[1387]{
   GP1:
	UF : 7, UT : 3,	CONFIG : 'F U T, 0, 1, 0',
	X =  -342.332  mm,	Y =    47.913  mm,	Z =     0.000  mm,
	W =  -167.380 deg,	P =    -0.011 deg,	R =   -83.337 deg
};
P[1388]{
   GP1:
	UF : 7, UT : 3,	CONFIG : 'F U T, 0, 1, 0',
	X =  -342.332  mm,	Y =    47.913  mm,	Z =     0.000  mm,
	W =  -167.380 deg,	P =    -0.011 deg,	R =   -83.337 deg
};
P[1389]{
   GP1:
	UF : 7, UT : 3,	CONFIG : 'F U T, 0, 1, 0',
	X =  -342.332  mm,	Y =    47.913  mm,	Z =     0.000  mm,
	W =  -167.380 deg,	P =    -0.011 deg,	R =   -83.337 deg
};
P[1390]{
   GP1:
	UF : 7, UT : 3,	CONFIG : 'F U T, 0, 1, 0',
	X =  -344.705  mm,	Y =    25.816  mm,	Z =     0.003  mm,
	W =  -167.372 deg,	P =    -0.002 deg,	R =   -79.244 deg
};
P[1391]{
   GP1:
	UF : 7, UT : 3,	CONFIG : 'F U T, 0, 1, 0',
	X =  -345.686  mm,	Y =     0.000  mm,	Z =     0.000  mm,
	W =  -167.361 deg,	P =     0.008 deg,	R =   -75.603 deg
};
P[1392]{
   GP1:
	UF : 7, UT : 3,	CONFIG : 'F U T, 0, 1, 0',
	X =  -345.686  mm,	Y =     0.000  mm,	Z =     0.000  mm,
	W =  -167.361 deg,	P =     0.008 deg,	R =   -75.603 deg
};
P[1393]{
   GP1:
	UF : 7, UT : 3,	CONFIG : 'F U T, 0, 1, 0',
	X =  -345.686  mm,	Y =     0.000  mm,	Z =     0.000  mm,
	W =  -167.361 deg,	P =     0.008 deg,	R =   -75.603 deg
};
P[1394]{
   GP1:
	UF : 7, UT : 3,	CONFIG : 'F U T, 0, 1, 0',
	X =  -345.686  mm,	Y =     0.000  mm,	Z =     0.000  mm,
	W =  -167.361 deg,	P =     0.008 deg,	R =   -75.603 deg
};
P[1395]{
   GP1:
	UF : 7, UT : 3,	CONFIG : 'F U T, 0, 1, 0',
	X =  -342.552  mm,	Y =     0.000  mm,	Z =     0.000  mm,
	W =  -167.361 deg,	P =     0.008 deg,	R =   -75.584 deg
};
P[1396]{
   GP1:
	UF : 7, UT : 3,	CONFIG : 'F U T, 0, 1, 0',
	X =  -342.552  mm,	Y =     0.000  mm,	Z =     0.000  mm,
	W =  -167.361 deg,	P =     0.008 deg,	R =   -75.584 deg
};
P[1397]{
   GP1:
	UF : 7, UT : 3,	CONFIG : 'F U T, 0, 1, 0',
	X =  -342.552  mm,	Y =     0.000  mm,	Z =     0.000  mm,
	W =  -167.361 deg,	P =     0.008 deg,	R =   -75.584 deg
};
P[1398]{
   GP1:
	UF : 7, UT : 3,	CONFIG : 'F U T, 0, 1, 0',
	X =  -342.552  mm,	Y =     0.000  mm,	Z =     0.000  mm,
	W =  -167.361 deg,	P =     0.008 deg,	R =   -75.584 deg
};
P[1399]{
   GP1:
	UF : 7, UT : 3,	CONFIG : 'F U T, 0, 1, 0',
	X =  -341.800  mm,	Y =    22.656  mm,	Z =     0.002  mm,
	W =  -167.370 deg,	P =    -0.001 deg,	R =   -78.735 deg
};
P[1400]{
   GP1:
	UF : 7, UT : 3,	CONFIG : 'F U T, 0, 1, 0',
	X =  -339.575  mm,	Y =    45.037  mm,	Z =     0.000  mm,
	W =  -167.378 deg,	P =    -0.011 deg,	R =   -81.919 deg
};
P[1401]{
   GP1:
	UF : 7, UT : 3,	CONFIG : 'F U T, 0, 1, 0',
	X =  -339.575  mm,	Y =    45.037  mm,	Z =     0.000  mm,
	W =  -167.378 deg,	P =    -0.011 deg,	R =   -81.919 deg
};
P[1402]{
   GP1:
	UF : 7, UT : 3,	CONFIG : 'F U T, 0, 1, 0',
	X =  -339.575  mm,	Y =    45.037  mm,	Z =     0.000  mm,
	W =  -167.378 deg,	P =    -0.011 deg,	R =   -81.919 deg
};
P[1403]{
   GP1:
	UF : 7, UT : 3,	CONFIG : 'F U T, 0, 1, 0',
	X =  -339.575  mm,	Y =    45.037  mm,	Z =     0.000  mm,
	W =  -167.378 deg,	P =    -0.011 deg,	R =   -81.919 deg
};
P[1404]{
   GP1:
	UF : 7, UT : 3,	CONFIG : 'F U T, 0, 0, 0',
	X =  -325.470  mm,	Y =   106.765  mm,	Z =     0.000  mm,
	W =  -167.618 deg,	P =     0.684 deg,	R =   -93.130 deg
};
P[1405]{
   GP1:
	UF : 7, UT : 3,	CONFIG : 'F U T, 0, 0, 0',
	X =  -325.470  mm,	Y =   106.765  mm,	Z =     0.000  mm,
	W =  -167.618 deg,	P =     0.684 deg,	R =   -93.130 deg
};
P[1406]{
   GP1:
	UF : 7, UT : 3,	CONFIG : 'F U T, 0, 0, 0',
	X =  -325.470  mm,	Y =   106.765  mm,	Z =     0.000  mm,
	W =  -167.618 deg,	P =     0.684 deg,	R =   -93.130 deg
};
P[1407]{
   GP1:
	UF : 7, UT : 3,	CONFIG : 'F U T, 0, 0, 0',
	X =  -325.470  mm,	Y =   106.765  mm,	Z =     0.000  mm,
	W =  -167.618 deg,	P =     0.684 deg,	R =   -93.130 deg
};
P[1408]{
   GP1:
	UF : 7, UT : 3,	CONFIG : 'F U T, 0, 0, 0',
	X =  -321.597  mm,	Y =   117.970  mm,	Z =     0.274  mm,
	W =  -167.697 deg,	P =     2.153 deg,	R =   -95.041 deg
};
P[1409]{
   GP1:
	UF : 7, UT : 3,	CONFIG : 'F U T, 0, 0, 0',
	X =  -320.331  mm,	Y =   121.319  mm,	Z =     0.406  mm,
	W =  -167.738 deg,	P =     2.368 deg,	R =   -95.784 deg
};
P[1410]{
   GP1:
	UF : 7, UT : 3,	CONFIG : 'F U T, 0, 0, 0',
	X =  -319.155  mm,	Y =   124.393  mm,	Z =     0.534  mm,
	W =  -167.774 deg,	P =     2.363 deg,	R =   -96.124 deg
};
P[1411]{
   GP1:
	UF : 7, UT : 3,	CONFIG : 'F U T, 0, 0, 0',
	X =  -317.879  mm,	Y =   127.633  mm,	Z =     0.663  mm,
	W =  -167.841 deg,	P =     2.145 deg,	R =   -96.813 deg
};
P[1412]{
   GP1:
	UF : 7, UT : 3,	CONFIG : 'F U T, 0, 0, 0',
	X =  -313.909  mm,	Y =   137.100  mm,	Z =     0.908  mm,
	W =  -168.040 deg,	P =     1.025 deg,	R =   -98.473 deg
};
P[1413]{
   GP1:
	UF : 7, UT : 3,	CONFIG : 'F U T, 0, 0, 0',
	X =  -307.714  mm,	Y =   150.492  mm,	Z =     0.986  mm,
	W =  -168.440 deg,	P =     0.127 deg,	R =  -100.987 deg
};
P[1414]{
   GP1:
	UF : 7, UT : 3,	CONFIG : 'F U T, 0, 0, 0',
	X =  -301.389  mm,	Y =   162.785  mm,	Z =     0.801  mm,
	W =  -168.743 deg,	P =    -1.086 deg,	R =  -103.380 deg
};
P[1415]{
   GP1:
	UF : 7, UT : 3,	CONFIG : 'F U T, 0, 0, 0',
	X =  -298.728  mm,	Y =   167.639  mm,	Z =     0.646  mm,
	W =  -168.684 deg,	P =    -1.479 deg,	R =  -104.289 deg
};
P[1416]{
   GP1:
	UF : 7, UT : 3,	CONFIG : 'F U T, 0, 0, 0',
	X =  -293.943  mm,	Y =   175.865  mm,	Z =     0.335  mm,
	W =  -168.467 deg,	P =    -1.585 deg,	R =  -105.877 deg
};
P[1417]{
   GP1:
	UF : 7, UT : 3,	CONFIG : 'F U T, 0, 0, 0',
	X =  -286.401  mm,	Y =   187.899  mm,	Z =     0.000  mm,
	W =  -168.114 deg,	P =    -0.620 deg,	R =  -108.438 deg
};
P[1418]{
   GP1:
	UF : 7, UT : 3,	CONFIG : 'F U T, 0, 0, 0',
	X =  -286.401  mm,	Y =   187.899  mm,	Z =     0.000  mm,
	W =  -168.114 deg,	P =    -0.620 deg,	R =  -108.438 deg
};
P[1419]{
   GP1:
	UF : 7, UT : 3,	CONFIG : 'F U T, 0, 0, 0',
	X =  -286.401  mm,	Y =   187.899  mm,	Z =     0.000  mm,
	W =  -168.114 deg,	P =    -0.620 deg,	R =  -108.438 deg
};
P[1420]{
   GP1:
	UF : 7, UT : 3,	CONFIG : 'F U T, 0, 0, 0',
	X =  -286.401  mm,	Y =   187.899  mm,	Z =     0.000  mm,
	W =  -168.114 deg,	P =    -0.620 deg,	R =  -108.438 deg
};
P[1421]{
   GP1:
	UF : 7, UT : 3,	CONFIG : 'F U T, 0, 0, 0',
	X =  -246.913  mm,	Y =   237.408  mm,	Z =     0.000  mm,
	W =  -167.403 deg,	P =     0.109 deg,	R =  -118.143 deg
};
P[1422]{
   GP1:
	UF : 7, UT : 3,	CONFIG : 'F U T, 0, 0, 0',
	X =  -246.913  mm,	Y =   237.408  mm,	Z =     0.000  mm,
	W =  -167.403 deg,	P =     0.109 deg,	R =  -118.143 deg
};
P[1423]{
   GP1:
	UF : 7, UT : 3,	CONFIG : 'F U T, 0, 0, 0',
	X =  -246.913  mm,	Y =   237.408  mm,	Z =     0.000  mm,
	W =  -167.403 deg,	P =     0.109 deg,	R =  -118.143 deg
};
P[1424]{
   GP1:
	UF : 7, UT : 3,	CONFIG : 'F U T, 0, 0, 0',
	X =  -246.913  mm,	Y =   237.408  mm,	Z =     0.000  mm,
	W =  -167.403 deg,	P =     0.109 deg,	R =  -118.143 deg
};
P[1425]{
   GP1:
	UF : 7, UT : 3,	CONFIG : 'F U T, 0, 0, 0',
	X =  -237.143  mm,	Y =   247.168  mm,	Z =     0.016  mm,
	W =  -167.390 deg,	P =     0.054 deg,	R =  -121.107 deg
};
P[1426]{
   GP1:
	UF : 7, UT : 3,	CONFIG : 'F U T, 0, 0, 0',
	X =  -225.839  mm,	Y =   257.537  mm,	Z =     0.019  mm,
	W =  -167.369 deg,	P =    -0.004 deg,	R =  -123.677 deg
};
P[1427]{
   GP1:
	UF : 7, UT : 3,	CONFIG : 'F U T, 0, 0, 0',
	X =  -210.011  mm,	Y =   270.610  mm,	Z =     0.013  mm,
	W =  -167.370 deg,	P =    -0.005 deg,	R =  -127.178 deg
};
P[1428]{
   GP1:
	UF : 7, UT : 3,	CONFIG : 'F U T, 0, 0, 0',
	X =  -193.044  mm,	Y =   282.962  mm,	Z =     0.005  mm,
	W =  -167.371 deg,	P =    -0.006 deg,	R =  -130.623 deg
};
P[1429]{
   GP1:
	UF : 7, UT : 3,	CONFIG : 'F U T, 0, 0, 0',
	X =  -176.512  mm,	Y =   293.549  mm,	Z =     0.000  mm,
	W =  -167.373 deg,	P =    -0.008 deg,	R =  -134.331 deg
};
P[1430]{
   GP1:
	UF : 7, UT : 3,	CONFIG : 'F U T, 0, 0, 0',
	X =  -176.512  mm,	Y =   293.549  mm,	Z =     0.000  mm,
	W =  -167.373 deg,	P =    -0.008 deg,	R =  -134.331 deg
};
P[1431]{
   GP1:
	UF : 7, UT : 3,	CONFIG : 'F U T, 0, 0, 0',
	X =  -176.512  mm,	Y =   293.549  mm,	Z =     0.000  mm,
	W =  -167.373 deg,	P =    -0.008 deg,	R =  -134.331 deg
};
P[1432]{
   GP1:
	UF : 7, UT : 3,	CONFIG : 'F U T, 0, 0, 0',
	X =  -176.512  mm,	Y =   293.549  mm,	Z =     0.000  mm,
	W =  -167.373 deg,	P =    -0.008 deg,	R =  -134.331 deg
};
P[1433]{
   GP1:
	UF : 7, UT : 3,	CONFIG : 'F U T, 0, 0, 0',
	X =  -119.466  mm,	Y =   321.037  mm,	Z =     0.000  mm,
	W =  -167.364 deg,	P =     0.002 deg,	R =  -144.809 deg
};
P[1434]{
   GP1:
	UF : 7, UT : 3,	CONFIG : 'F U T, 0, 0, 0',
	X =  -119.466  mm,	Y =   321.037  mm,	Z =     0.000  mm,
	W =  -167.364 deg,	P =     0.002 deg,	R =  -144.809 deg
};
P[1435]{
   GP1:
	UF : 7, UT : 3,	CONFIG : 'F U T, 0, 0, 0',
	X =  -119.466  mm,	Y =   321.037  mm,	Z =     0.000  mm,
	W =  -167.364 deg,	P =     0.002 deg,	R =  -144.809 deg
};
P[1436]{
   GP1:
	UF : 7, UT : 3,	CONFIG : 'F U T, 0, 0, 0',
	X =  -119.466  mm,	Y =   321.037  mm,	Z =     0.000  mm,
	W =  -167.364 deg,	P =     0.002 deg,	R =  -144.809 deg
};
P[1437]{
   GP1:
	UF : 7, UT : 3,	CONFIG : 'F U T, 0, 0, 0',
	X =   -97.811  mm,	Y =   328.281  mm,	Z =     0.000  mm,
	W =  -167.364 deg,	P =     0.002 deg,	R =  -148.325 deg
};
P[1438]{
   GP1:
	UF : 7, UT : 3,	CONFIG : 'F U T, 0, 0, 0',
	X =   -76.713  mm,	Y =   333.844  mm,	Z =     0.000  mm,
	W =  -167.364 deg,	P =     0.001 deg,	R =  -151.969 deg
};
P[1439]{
   GP1:
	UF : 7, UT : 3,	CONFIG : 'F U T, 0, 0, 0',
	X =   -55.045  mm,	Y =   338.083  mm,	Z =     0.000  mm,
	W =  -167.364 deg,	P =     0.000 deg,	R =  -155.603 deg
};
P[1440]{
   GP1:
	UF : 7, UT : 3,	CONFIG : 'F U T, 0, 0, 0',
	X =   -31.661  mm,	Y =   341.073  mm,	Z =     0.000  mm,
	W =  -167.364 deg,	P =     0.000 deg,	R =  -159.256 deg
};
P[1441]{
   GP1:
	UF : 7, UT : 3,	CONFIG : 'F U T, 0, 0, 0',
	X =   -31.661  mm,	Y =   341.073  mm,	Z =     0.000  mm,
	W =  -167.364 deg,	P =     0.000 deg,	R =  -159.256 deg
};
P[1442]{
   GP1:
	UF : 7, UT : 3,	CONFIG : 'F U T, 0, 0, 0',
	X =   -31.661  mm,	Y =   341.073  mm,	Z =     0.000  mm,
	W =  -167.364 deg,	P =     0.000 deg,	R =  -159.256 deg
};
P[1443]{
   GP1:
	UF : 7, UT : 3,	CONFIG : 'F U T, 0, 0, 0',
	X =   -31.661  mm,	Y =   341.073  mm,	Z =     0.000  mm,
	W =  -167.364 deg,	P =     0.000 deg,	R =  -159.256 deg
};
P[1444]{
   GP1:
	UF : 7, UT : 3,	CONFIG : 'F U T, 0, 0, 0',
	X =    31.661  mm,	Y =   341.073  mm,	Z =     0.000  mm,
	W =  -167.363 deg,	P =     0.000 deg,	R =  -170.633 deg
};
P[1445]{
   GP1:
	UF : 7, UT : 3,	CONFIG : 'F U T, 0, 0, 0',
	X =    31.661  mm,	Y =   341.073  mm,	Z =     0.000  mm,
	W =  -167.363 deg,	P =     0.000 deg,	R =  -170.633 deg
};
P[1446]{
   GP1:
	UF : 7, UT : 3,	CONFIG : 'F U T, 0, 0, 0',
	X =    31.661  mm,	Y =   341.073  mm,	Z =     0.000  mm,
	W =  -167.363 deg,	P =     0.000 deg,	R =  -170.633 deg
};
P[1447]{
   GP1:
	UF : 7, UT : 3,	CONFIG : 'F U T, 0, 0, 0',
	X =    31.661  mm,	Y =   341.073  mm,	Z =     0.000  mm,
	W =  -167.363 deg,	P =     0.000 deg,	R =  -170.633 deg
};
P[1448]{
   GP1:
	UF : 7, UT : 3,	CONFIG : 'F U T, 0, 0, 0',
	X =    55.044  mm,	Y =   338.083  mm,	Z =     0.000  mm,
	W =  -167.364 deg,	P =     0.000 deg,	R =  -174.259 deg
};
P[1449]{
   GP1:
	UF : 7, UT : 3,	CONFIG : 'F U T, 0, 0, 0',
	X =    76.579  mm,	Y =   333.872  mm,	Z =     0.000  mm,
	W =  -167.364 deg,	P =     0.000 deg,	R =  -177.903 deg
};
P[1450]{
   GP1:
	UF : 7, UT : 3,	CONFIG : 'F U T, 0, 0, 0',
	X =    97.701  mm,	Y =   328.313  mm,	Z =     0.000  mm,
	W =  -167.364 deg,	P =     0.000 deg,	R =   178.462 deg
};
P[1451]{
   GP1:
	UF : 7, UT : 3,	CONFIG : 'F U T, 0, 0, 0',
	X =   119.466  mm,	Y =   321.037  mm,	Z =     0.000  mm,
	W =  -167.364 deg,	P =     0.000 deg,	R =   174.931 deg
};
P[1452]{
   GP1:
	UF : 7, UT : 3,	CONFIG : 'F U T, 0, 0, 0',
	X =   119.466  mm,	Y =   321.037  mm,	Z =     0.000  mm,
	W =  -167.364 deg,	P =     0.000 deg,	R =   174.931 deg
};
P[1453]{
   GP1:
	UF : 7, UT : 3,	CONFIG : 'F U T, 0, 0, 0',
	X =   119.466  mm,	Y =   321.037  mm,	Z =     0.000  mm,
	W =  -167.364 deg,	P =     0.000 deg,	R =   174.931 deg
};
P[1454]{
   GP1:
	UF : 7, UT : 3,	CONFIG : 'F U T, 0, 0, 0',
	X =   119.466  mm,	Y =   321.037  mm,	Z =     0.000  mm,
	W =  -167.364 deg,	P =     0.000 deg,	R =   174.931 deg
};
P[1455]{
   GP1:
	UF : 7, UT : 3,	CONFIG : 'F U T, 0, 0, 0',
	X =   176.512  mm,	Y =   293.549  mm,	Z =     0.000  mm,
	W =  -167.364 deg,	P =     0.001 deg,	R =   164.499 deg
};
P[1456]{
   GP1:
	UF : 7, UT : 3,	CONFIG : 'F U T, 0, 0, 0',
	X =   176.512  mm,	Y =   293.549  mm,	Z =     0.000  mm,
	W =  -167.364 deg,	P =     0.001 deg,	R =   164.499 deg
};
P[1457]{
   GP1:
	UF : 7, UT : 3,	CONFIG : 'F U T, 0, 0, 0',
	X =   176.512  mm,	Y =   293.549  mm,	Z =     0.000  mm,
	W =  -167.364 deg,	P =     0.001 deg,	R =   164.499 deg
};
P[1458]{
   GP1:
	UF : 7, UT : 3,	CONFIG : 'F U T, 0, 0, 0',
	X =   176.512  mm,	Y =   293.549  mm,	Z =     0.000  mm,
	W =  -167.364 deg,	P =     0.001 deg,	R =   164.499 deg
};
P[1459]{
   GP1:
	UF : 7, UT : 3,	CONFIG : 'F U T, 0, 0, 0',
	X =   194.879  mm,	Y =   281.695  mm,	Z =     0.000  mm,
	W =  -167.364 deg,	P =     0.000 deg,	R =   160.317 deg
};
P[1460]{
   GP1:
	UF : 7, UT : 3,	CONFIG : 'F U T, 0, 0, 0',
	X =   213.593  mm,	Y =   267.780  mm,	Z =     0.001  mm,
	W =  -167.364 deg,	P =     0.000 deg,	R =   156.430 deg
};
P[1461]{
   GP1:
	UF : 7, UT : 3,	CONFIG : 'F U T, 0, 0, 0',
	X =   231.580  mm,	Y =   252.386  mm,	Z =     0.000  mm,
	W =  -167.365 deg,	P =    -0.001 deg,	R =   152.593 deg
};
P[1462]{
   GP1:
	UF : 7, UT : 3,	CONFIG : 'F U T, 0, 0, 0',
	X =   246.913  mm,	Y =   237.408  mm,	Z =     0.000  mm,
	W =  -167.365 deg,	P =    -0.001 deg,	R =   148.257 deg
};
P[1463]{
   GP1:
	UF : 7, UT : 3,	CONFIG : 'F U T, 0, 0, 0',
	X =   246.913  mm,	Y =   237.408  mm,	Z =     0.000  mm,
	W =  -167.365 deg,	P =    -0.001 deg,	R =   148.257 deg
};
P[1464]{
   GP1:
	UF : 7, UT : 3,	CONFIG : 'F U T, 0, 0, 0',
	X =   246.913  mm,	Y =   237.408  mm,	Z =     0.000  mm,
	W =  -167.365 deg,	P =    -0.001 deg,	R =   148.257 deg
};
P[1465]{
   GP1:
	UF : 7, UT : 3,	CONFIG : 'F U T, 0, 0, 0',
	X =   246.913  mm,	Y =   237.408  mm,	Z =     0.000  mm,
	W =  -167.365 deg,	P =    -0.001 deg,	R =   148.257 deg
};
P[1466]{
   GP1:
	UF : 7, UT : 3,	CONFIG : 'F U T, 0, 0, 0',
	X =   286.401  mm,	Y =   187.899  mm,	Z =     0.000  mm,
	W =  -167.364 deg,	P =     0.001 deg,	R =   138.566 deg
};
P[1467]{
   GP1:
	UF : 7, UT : 3,	CONFIG : 'F U T, 0, 0, 0',
	X =   286.401  mm,	Y =   187.899  mm,	Z =     0.000  mm,
	W =  -167.364 deg,	P =     0.001 deg,	R =   138.566 deg
};
P[1468]{
   GP1:
	UF : 7, UT : 3,	CONFIG : 'F U T, 0, 0, 0',
	X =   286.401  mm,	Y =   187.899  mm,	Z =     0.000  mm,
	W =  -167.364 deg,	P =     0.001 deg,	R =   138.566 deg
};
P[1469]{
   GP1:
	UF : 7, UT : 3,	CONFIG : 'F U T, 0, 0, 0',
	X =   286.401  mm,	Y =   187.899  mm,	Z =     0.000  mm,
	W =  -167.364 deg,	P =     0.001 deg,	R =   138.566 deg
};
P[1470]{
   GP1:
	UF : 7, UT : 3,	CONFIG : 'F U T, 0, 0, 0',
	X =   297.955  mm,	Y =   168.979  mm,	Z =     0.000  mm,
	W =  -167.364 deg,	P =     0.001 deg,	R =   134.646 deg
};
P[1471]{
   GP1:
	UF : 7, UT : 3,	CONFIG : 'F U T, 0, 0, 0',
	X =   308.551  mm,	Y =   148.749  mm,	Z =     0.000  mm,
	W =  -167.365 deg,	P =     0.000 deg,	R =   130.867 deg
};
P[1472]{
   GP1:
	UF : 7, UT : 3,	CONFIG : 'F U T, 0, 0, 0',
	X =   317.654  mm,	Y =   128.171  mm,	Z =     0.000  mm,
	W =  -167.365 deg,	P =     0.000 deg,	R =   127.061 deg
};
P[1473]{
   GP1:
	UF : 7, UT : 3,	CONFIG : 'F U T, 0, 0, 0',
	X =   325.470  mm,	Y =   106.765  mm,	Z =     0.000  mm,
	W =  -167.365 deg,	P =    -0.001 deg,	R =   123.242 deg
};
P[1474]{
   GP1:
	UF : 7, UT : 3,	CONFIG : 'F U T, 0, 0, 0',
	X =   325.470  mm,	Y =   106.765  mm,	Z =     0.000  mm,
	W =  -167.365 deg,	P =    -0.001 deg,	R =   123.242 deg
};
P[1475]{
   GP1:
	UF : 7, UT : 3,	CONFIG : 'F U T, 0, 0, 0',
	X =   325.470  mm,	Y =   106.765  mm,	Z =     0.000  mm,
	W =  -167.365 deg,	P =    -0.001 deg,	R =   123.242 deg
};
P[1476]{
   GP1:
	UF : 7, UT : 3,	CONFIG : 'F U T, 0, 0, 0',
	X =   325.470  mm,	Y =   106.765  mm,	Z =     0.000  mm,
	W =  -167.365 deg,	P =    -0.001 deg,	R =   123.242 deg
};
P[1477]{
   GP1:
	UF : 7, UT : 3,	CONFIG : 'F U T, 0, 0, 0',
	X =   339.575  mm,	Y =    45.037  mm,	Z =     0.000  mm,
	W =  -167.364 deg,	P =     0.001 deg,	R =   112.025 deg
};
P[1478]{
   GP1:
	UF : 7, UT : 3,	CONFIG : 'F U T, 0, 0, 0',
	X =   339.575  mm,	Y =    45.037  mm,	Z =     0.000  mm,
	W =  -167.364 deg,	P =     0.001 deg,	R =   112.025 deg
};
P[1479]{
   GP1:
	UF : 7, UT : 3,	CONFIG : 'F U T, 0, 0, 0',
	X =   339.575  mm,	Y =    45.037  mm,	Z =     0.000  mm,
	W =  -167.364 deg,	P =     0.001 deg,	R =   112.025 deg
};
P[1480]{
   GP1:
	UF : 7, UT : 3,	CONFIG : 'F U T, 0, 0, 0',
	X =   339.575  mm,	Y =    45.037  mm,	Z =     0.000  mm,
	W =  -167.364 deg,	P =     0.001 deg,	R =   112.025 deg
};
P[1481]{
   GP1:
	UF : 7, UT : 3,	CONFIG : 'F U T, 0, 0, 0',
	X =   341.816  mm,	Y =    22.422  mm,	Z =     0.000  mm,
	W =  -167.364 deg,	P =     0.000 deg,	R =   108.791 deg
};
P[1482]{
   GP1:
	UF : 7, UT : 3,	CONFIG : 'F U T, 0, 0, 0',
	X =   342.552  mm,	Y =     0.000  mm,	Z =     0.000  mm,
	W =  -167.364 deg,	P =    -0.001 deg,	R =   105.698 deg
};
P[1483]{
   GP1:
	UF : 7, UT : 3,	CONFIG : 'F U T, 0, 0, 0',
	X =   342.552  mm,	Y =     0.000  mm,	Z =     0.000  mm,
	W =  -167.364 deg,	P =    -0.001 deg,	R =   105.698 deg
};
P[1484]{
   GP1:
	UF : 7, UT : 3,	CONFIG : 'F U T, 0, 0, 0',
	X =   342.552  mm,	Y =     0.000  mm,	Z =     0.000  mm,
	W =  -167.364 deg,	P =    -0.001 deg,	R =   105.698 deg
};
P[1485]{
   GP1:
	UF : 7, UT : 3,	CONFIG : 'F U T, 0, 0, 0',
	X =   342.552  mm,	Y =     0.000  mm,	Z =     0.000  mm,
	W =  -167.364 deg,	P =    -0.001 deg,	R =   105.698 deg
};
P[1486]{
   GP1:
	UF : 7, UT : 3,	CONFIG : 'F U T, 0, 0, 0',
	X =   339.418  mm,	Y =     0.000  mm,	Z =     0.000  mm,
	W =  -167.364 deg,	P =    -0.001 deg,	R =   105.695 deg
};
P[1487]{
   GP1:
	UF : 7, UT : 3,	CONFIG : 'F U T, 0, 0, 0',
	X =   339.418  mm,	Y =     0.000  mm,	Z =     0.000  mm,
	W =  -167.364 deg,	P =    -0.001 deg,	R =   105.695 deg
};
P[1488]{
   GP1:
	UF : 7, UT : 3,	CONFIG : 'F U T, 0, 0, 0',
	X =   339.418  mm,	Y =     0.000  mm,	Z =     0.000  mm,
	W =  -167.364 deg,	P =    -0.001 deg,	R =   105.695 deg
};
P[1489]{
   GP1:
	UF : 7, UT : 3,	CONFIG : 'F U T, 0, 0, 0',
	X =   339.418  mm,	Y =     0.000  mm,	Z =     0.000  mm,
	W =  -167.364 deg,	P =    -0.001 deg,	R =   105.695 deg
};
P[1490]{
   GP1:
	UF : 7, UT : 3,	CONFIG : 'F U T, 0, 0, 0',
	X =   338.647  mm,	Y =    22.681  mm,	Z =     0.000  mm,
	W =  -167.364 deg,	P =     0.000 deg,	R =   108.893 deg
};
P[1491]{
   GP1:
	UF : 7, UT : 3,	CONFIG : 'F U T, 0, 0, 0',
	X =   336.714  mm,	Y =    42.617  mm,	Z =     0.000  mm,
	W =  -167.364 deg,	P =     0.001 deg,	R =   112.211 deg
};
P[1492]{
   GP1:
	UF : 7, UT : 3,	CONFIG : 'F U T, 0, 0, 0',
	X =   336.714  mm,	Y =    42.617  mm,	Z =     0.000  mm,
	W =  -167.364 deg,	P =     0.001 deg,	R =   112.211 deg
};
P[1493]{
   GP1:
	UF : 7, UT : 3,	CONFIG : 'F U T, 0, 0, 0',
	X =   336.714  mm,	Y =    42.617  mm,	Z =     0.000  mm,
	W =  -167.364 deg,	P =     0.001 deg,	R =   112.211 deg
};
P[1494]{
   GP1:
	UF : 7, UT : 3,	CONFIG : 'F U T, 0, 0, 0',
	X =   336.714  mm,	Y =    42.617  mm,	Z =     0.000  mm,
	W =  -167.364 deg,	P =     0.001 deg,	R =   112.211 deg
};
P[1495]{
   GP1:
	UF : 7, UT : 3,	CONFIG : 'F U T, 0, 0, 0',
	X =   321.857  mm,	Y =   107.699  mm,	Z =     0.000  mm,
	W =  -167.365 deg,	P =    -0.001 deg,	R =   122.977 deg
};
P[1496]{
   GP1:
	UF : 7, UT : 3,	CONFIG : 'F U T, 0, 0, 0',
	X =   321.857  mm,	Y =   107.699  mm,	Z =     0.000  mm,
	W =  -167.365 deg,	P =    -0.001 deg,	R =   122.977 deg
};
P[1497]{
   GP1:
	UF : 7, UT : 3,	CONFIG : 'F U T, 0, 0, 0',
	X =   321.857  mm,	Y =   107.699  mm,	Z =     0.000  mm,
	W =  -167.365 deg,	P =    -0.001 deg,	R =   122.977 deg
};
P[1498]{
   GP1:
	UF : 7, UT : 3,	CONFIG : 'F U T, 0, 0, 0',
	X =   321.857  mm,	Y =   107.699  mm,	Z =     0.000  mm,
	W =  -167.365 deg,	P =    -0.001 deg,	R =   122.977 deg
};
P[1499]{
   GP1:
	UF : 7, UT : 3,	CONFIG : 'F U T, 0, 0, 0',
	X =   315.156  mm,	Y =   125.993  mm,	Z =     0.000  mm,
	W =  -167.365 deg,	P =    -0.001 deg,	R =   126.868 deg
};
P[1500]{
   GP1:
	UF : 7, UT : 3,	CONFIG : 'F U T, 0, 0, 0',
	X =   306.745  mm,	Y =   145.278  mm,	Z =     0.000  mm,
	W =  -167.365 deg,	P =     0.000 deg,	R =   130.396 deg
};
P[1501]{
   GP1:
	UF : 7, UT : 3,	CONFIG : 'F U T, 0, 0, 0',
	X =   297.052  mm,	Y =   164.179  mm,	Z =     0.000  mm,
	W =  -167.364 deg,	P =     0.001 deg,	R =   133.923 deg
};
P[1502]{
   GP1:
	UF : 7, UT : 3,	CONFIG : 'F U T, 0, 0, 0',
	X =   284.886  mm,	Y =   184.508  mm,	Z =     0.000  mm,
	W =  -167.364 deg,	P =     0.001 deg,	R =   137.383 deg
};
P[1503]{
   GP1:
	UF : 7, UT : 3,	CONFIG : 'F U T, 0, 0, 0',
	X =   284.886  mm,	Y =   184.508  mm,	Z =     0.000  mm,
	W =  -167.364 deg,	P =     0.001 deg,	R =   137.383 deg
};
P[1504]{
   GP1:
	UF : 7, UT : 3,	CONFIG : 'F U T, 0, 0, 0',
	X =   284.886  mm,	Y =   184.508  mm,	Z =     0.000  mm,
	W =  -167.364 deg,	P =     0.001 deg,	R =   137.383 deg
};
P[1505]{
   GP1:
	UF : 7, UT : 3,	CONFIG : 'F U T, 0, 0, 0',
	X =   284.886  mm,	Y =   184.508  mm,	Z =     0.000  mm,
	W =  -167.364 deg,	P =     0.001 deg,	R =   137.383 deg
};
P[1506]{
   GP1:
	UF : 7, UT : 3,	CONFIG : 'F U T, 0, 0, 0',
	X =   243.267  mm,	Y =   236.685  mm,	Z =     0.000  mm,
	W =  -167.365 deg,	P =    -0.001 deg,	R =   149.492 deg
};
P[1507]{
   GP1:
	UF : 7, UT : 3,	CONFIG : 'F U T, 0, 0, 0',
	X =   243.267  mm,	Y =   236.685  mm,	Z =     0.000  mm,
	W =  -167.365 deg,	P =    -0.001 deg,	R =   149.492 deg
};
P[1508]{
   GP1:
	UF : 7, UT : 3,	CONFIG : 'F U T, 0, 0, 0',
	X =   243.267  mm,	Y =   236.685  mm,	Z =     0.000  mm,
	W =  -167.365 deg,	P =    -0.001 deg,	R =   149.492 deg
};
P[1509]{
   GP1:
	UF : 7, UT : 3,	CONFIG : 'F U T, 0, 0, 0',
	X =   243.267  mm,	Y =   236.685  mm,	Z =     0.000  mm,
	W =  -167.365 deg,	P =    -0.001 deg,	R =   149.492 deg
};
P[1510]{
   GP1:
	UF : 7, UT : 3,	CONFIG : 'F U T, 0, 0, 0',
	X =   227.208  mm,	Y =   252.135  mm,	Z =     0.001  mm,
	W =  -167.365 deg,	P =    -0.001 deg,	R =   152.973 deg
};
P[1511]{
   GP1:
	UF : 7, UT : 3,	CONFIG : 'F U T, 0, 0, 0',
	X =   210.955  mm,	Y =   265.877  mm,	Z =     0.001  mm,
	W =  -167.364 deg,	P =     0.000 deg,	R =   156.582 deg
};
P[1512]{
   GP1:
	UF : 7, UT : 3,	CONFIG : 'F U T, 0, 0, 0',
	X =   193.925  mm,	Y =   278.540  mm,	Z =     0.000  mm,
	W =  -167.364 deg,	P =     0.000 deg,	R =   160.209 deg
};
P[1513]{
   GP1:
	UF : 7, UT : 3,	CONFIG : 'F U T, 0, 0, 0',
	X =   176.618  mm,	Y =   289.827  mm,	Z =     0.000  mm,
	W =  -167.364 deg,	P =     0.001 deg,	R =   163.961 deg
};
P[1514]{
   GP1:
	UF : 7, UT : 3,	CONFIG : 'F U T, 0, 0, 0',
	X =   176.618  mm,	Y =   289.827  mm,	Z =     0.000  mm,
	W =  -167.364 deg,	P =     0.001 deg,	R =   163.961 deg
};
P[1515]{
   GP1:
	UF : 7, UT : 3,	CONFIG : 'F U T, 0, 0, 0',
	X =   176.618  mm,	Y =   289.827  mm,	Z =     0.000  mm,
	W =  -167.364 deg,	P =     0.001 deg,	R =   163.961 deg
};
P[1516]{
   GP1:
	UF : 7, UT : 3,	CONFIG : 'F U T, 0, 0, 0',
	X =   176.618  mm,	Y =   289.827  mm,	Z =     0.000  mm,
	W =  -167.364 deg,	P =     0.001 deg,	R =   163.961 deg
};
P[1517]{
   GP1:
	UF : 7, UT : 3,	CONFIG : 'F U T, 0, 0, 0',
	X =   116.480  mm,	Y =   318.793  mm,	Z =     0.000  mm,
	W =  -167.364 deg,	P =     0.000 deg,	R =   175.343 deg
};
P[1518]{
   GP1:
	UF : 7, UT : 3,	CONFIG : 'F U T, 0, 0, 0',
	X =   116.480  mm,	Y =   318.793  mm,	Z =     0.000  mm,
	W =  -167.364 deg,	P =     0.000 deg,	R =   175.343 deg
};
P[1519]{
   GP1:
	UF : 7, UT : 3,	CONFIG : 'F U T, 0, 0, 0',
	X =   116.480  mm,	Y =   318.793  mm,	Z =     0.000  mm,
	W =  -167.364 deg,	P =     0.000 deg,	R =   175.343 deg
};
P[1520]{
   GP1:
	UF : 7, UT : 3,	CONFIG : 'F U T, 0, 0, 0',
	X =   116.480  mm,	Y =   318.793  mm,	Z =     0.000  mm,
	W =  -167.364 deg,	P =     0.000 deg,	R =   175.343 deg
};
P[1521]{
   GP1:
	UF : 7, UT : 3,	CONFIG : 'F U T, 0, 0, 0',
	X =    95.046  mm,	Y =   325.832  mm,	Z =     0.000  mm,
	W =  -167.364 deg,	P =     0.000 deg,	R =   178.833 deg
};
P[1522]{
   GP1:
	UF : 7, UT : 3,	CONFIG : 'F U T, 0, 0, 0',
	X =    74.334  mm,	Y =   331.167  mm,	Z =     0.000  mm,
	W =  -167.364 deg,	P =     0.000 deg,	R =  -177.594 deg
};
P[1523]{
   GP1:
	UF : 7, UT : 3,	CONFIG : 'F U T, 0, 0, 0',
	X =    53.315  mm,	Y =   335.191  mm,	Z =     0.000  mm,
	W =  -167.364 deg,	P =     0.000 deg,	R =  -174.020 deg
};
P[1524]{
   GP1:
	UF : 7, UT : 3,	CONFIG : 'F U T, 0, 0, 0',
	X =    33.379  mm,	Y =   337.752  mm,	Z =     0.000  mm,
	W =  -167.363 deg,	P =     0.000 deg,	R =  -170.212 deg
};
P[1525]{
   GP1:
	UF : 7, UT : 3,	CONFIG : 'F U T, 0, 0, 0',
	X =    33.379  mm,	Y =   337.752  mm,	Z =     0.000  mm,
	W =  -167.363 deg,	P =     0.000 deg,	R =  -170.212 deg
};
P[1526]{
   GP1:
	UF : 7, UT : 3,	CONFIG : 'F U T, 0, 0, 0',
	X =    33.379  mm,	Y =   337.752  mm,	Z =     0.000  mm,
	W =  -167.363 deg,	P =     0.000 deg,	R =  -170.212 deg
};
P[1527]{
   GP1:
	UF : 7, UT : 3,	CONFIG : 'F U T, 0, 0, 0',
	X =    33.379  mm,	Y =   337.752  mm,	Z =     0.000  mm,
	W =  -167.363 deg,	P =     0.000 deg,	R =  -170.212 deg
};
P[1528]{
   GP1:
	UF : 7, UT : 3,	CONFIG : 'F U T, 0, 0, 0',
	X =   -33.379  mm,	Y =   337.752  mm,	Z =     0.000  mm,
	W =  -167.364 deg,	P =     0.000 deg,	R =  -159.668 deg
};
P[1529]{
   GP1:
	UF : 7, UT : 3,	CONFIG : 'F U T, 0, 0, 0',
	X =   -33.379  mm,	Y =   337.752  mm,	Z =     0.000  mm,
	W =  -167.364 deg,	P =     0.000 deg,	R =  -159.668 deg
};
P[1530]{
   GP1:
	UF : 7, UT : 3,	CONFIG : 'F U T, 0, 0, 0',
	X =   -33.379  mm,	Y =   337.752  mm,	Z =     0.000  mm,
	W =  -167.364 deg,	P =     0.000 deg,	R =  -159.668 deg
};
P[1531]{
   GP1:
	UF : 7, UT : 3,	CONFIG : 'F U T, 0, 0, 0',
	X =   -33.379  mm,	Y =   337.752  mm,	Z =     0.000  mm,
	W =  -167.364 deg,	P =     0.000 deg,	R =  -159.668 deg
};
P[1532]{
   GP1:
	UF : 7, UT : 3,	CONFIG : 'F U T, 0, 0, 0',
	X =   -53.168  mm,	Y =   335.215  mm,	Z =     0.000  mm,
	W =  -167.364 deg,	P =     0.000 deg,	R =  -155.903 deg
};
P[1533]{
   GP1:
	UF : 7, UT : 3,	CONFIG : 'F U T, 0, 0, 0',
	X =   -74.023  mm,	Y =   331.235  mm,	Z =     0.000  mm,
	W =  -167.364 deg,	P =     0.001 deg,	R =  -152.367 deg
};
P[1534]{
   GP1:
	UF : 7, UT : 3,	CONFIG : 'F U T, 0, 0, 0',
	X =   -94.595  mm,	Y =   325.959  mm,	Z =     0.000  mm,
	W =  -167.364 deg,	P =     0.002 deg,	R =  -148.827 deg
};
P[1535]{
   GP1:
	UF : 7, UT : 3,	CONFIG : 'F U T, 0, 0, 0',
	X =  -116.480  mm,	Y =   318.793  mm,	Z =     0.000  mm,
	W =  -167.364 deg,	P =     0.002 deg,	R =  -145.310 deg
};
P[1536]{
   GP1:
	UF : 7, UT : 3,	CONFIG : 'F U T, 0, 0, 0',
	X =  -116.480  mm,	Y =   318.793  mm,	Z =     0.000  mm,
	W =  -167.364 deg,	P =     0.002 deg,	R =  -145.310 deg
};
P[1537]{
   GP1:
	UF : 7, UT : 3,	CONFIG : 'F U T, 0, 0, 0',
	X =  -116.480  mm,	Y =   318.793  mm,	Z =     0.000  mm,
	W =  -167.364 deg,	P =     0.002 deg,	R =  -145.310 deg
};
P[1538]{
   GP1:
	UF : 7, UT : 3,	CONFIG : 'F U T, 0, 0, 0',
	X =  -116.480  mm,	Y =   318.793  mm,	Z =     0.000  mm,
	W =  -167.364 deg,	P =     0.002 deg,	R =  -145.310 deg
};
P[1539]{
   GP1:
	UF : 7, UT : 3,	CONFIG : 'F U T, 0, 0, 0',
	X =  -176.618  mm,	Y =   289.827  mm,	Z =     0.000  mm,
	W =  -167.372 deg,	P =    -0.009 deg,	R =  -133.843 deg
};
P[1540]{
   GP1:
	UF : 7, UT : 3,	CONFIG : 'F U T, 0, 0, 0',
	X =  -176.618  mm,	Y =   289.827  mm,	Z =     0.000  mm,
	W =  -167.372 deg,	P =    -0.009 deg,	R =  -133.843 deg
};
P[1541]{
   GP1:
	UF : 7, UT : 3,	CONFIG : 'F U T, 0, 0, 0',
	X =  -176.618  mm,	Y =   289.827  mm,	Z =     0.000  mm,
	W =  -167.372 deg,	P =    -0.009 deg,	R =  -133.843 deg
};
P[1542]{
   GP1:
	UF : 7, UT : 3,	CONFIG : 'F U T, 0, 0, 0',
	X =  -176.618  mm,	Y =   289.827  mm,	Z =     0.000  mm,
	W =  -167.372 deg,	P =    -0.009 deg,	R =  -133.843 deg
};
P[1543]{
   GP1:
	UF : 7, UT : 3,	CONFIG : 'F U T, 0, 0, 0',
	X =  -192.066  mm,	Y =   279.834  mm,	Z =     0.005  mm,
	W =  -167.371 deg,	P =    -0.008 deg,	R =  -130.435 deg
};
P[1544]{
   GP1:
	UF : 7, UT : 3,	CONFIG : 'F U T, 0, 0, 0',
	X =  -207.852  mm,	Y =   268.316  mm,	Z =     0.013  mm,
	W =  -167.368 deg,	P =    -0.007 deg,	R =  -127.234 deg
};
P[1545]{
   GP1:
	UF : 7, UT : 3,	CONFIG : 'F U T, 0, 0, 0',
	X =  -222.508  mm,	Y =   256.289  mm,	Z =     0.019  mm,
	W =  -167.366 deg,	P =    -0.006 deg,	R =  -123.956 deg
};
P[1546]{
   GP1:
	UF : 7, UT : 3,	CONFIG : 'F U T, 0, 0, 0',
	X =  -232.839  mm,	Y =   246.952  mm,	Z =     0.016  mm,
	W =  -167.382 deg,	P =     0.050 deg,	R =  -121.608 deg
};
P[1547]{
   GP1:
	UF : 7, UT : 3,	CONFIG : 'F U T, 0, 0, 0',
	X =  -243.267  mm,	Y =   236.685  mm,	Z =     0.000  mm,
	W =  -167.393 deg,	P =     0.110 deg,	R =  -119.381 deg
};
P[1548]{
   GP1:
	UF : 7, UT : 3,	CONFIG : 'F U T, 0, 0, 0',
	X =  -243.267  mm,	Y =   236.685  mm,	Z =     0.000  mm,
	W =  -167.393 deg,	P =     0.110 deg,	R =  -119.381 deg
};
P[1549]{
   GP1:
	UF : 7, UT : 3,	CONFIG : 'F U T, 0, 0, 0',
	X =  -243.267  mm,	Y =   236.685  mm,	Z =     0.000  mm,
	W =  -167.393 deg,	P =     0.110 deg,	R =  -119.381 deg
};
P[1550]{
   GP1:
	UF : 7, UT : 3,	CONFIG : 'F U T, 0, 0, 0',
	X =  -243.267  mm,	Y =   236.685  mm,	Z =     0.000  mm,
	W =  -167.393 deg,	P =     0.110 deg,	R =  -119.381 deg
};
P[1551]{
   GP1:
	UF : 7, UT : 3,	CONFIG : 'F U T, 0, 0, 0',
	X =  -284.886  mm,	Y =   184.508  mm,	Z =     0.000  mm,
	W =  -168.146 deg,	P =    -0.761 deg,	R =  -107.268 deg
};
P[1552]{
   GP1:
	UF : 7, UT : 3,	CONFIG : 'F U T, 0, 0, 0',
	X =  -284.886  mm,	Y =   184.508  mm,	Z =     0.000  mm,
	W =  -168.146 deg,	P =    -0.761 deg,	R =  -107.268 deg
};
P[1553]{
   GP1:
	UF : 7, UT : 3,	CONFIG : 'F U T, 0, 0, 0',
	X =  -284.886  mm,	Y =   184.508  mm,	Z =     0.000  mm,
	W =  -168.146 deg,	P =    -0.761 deg,	R =  -107.268 deg
};
P[1554]{
   GP1:
	UF : 7, UT : 3,	CONFIG : 'F U T, 0, 0, 0',
	X =  -284.886  mm,	Y =   184.508  mm,	Z =     0.000  mm,
	W =  -168.146 deg,	P =    -0.761 deg,	R =  -107.268 deg
};
P[1555]{
   GP1:
	UF : 7, UT : 3,	CONFIG : 'F U T, 0, 0, 0',
	X =  -289.407  mm,	Y =   177.311  mm,	Z =     0.192  mm,
	W =  -168.363 deg,	P =    -1.395 deg,	R =  -106.397 deg
};
P[1556]{
   GP1:
	UF : 7, UT : 3,	CONFIG : 'F U T, 0, 0, 0',
	X =  -292.004  mm,	Y =   173.005  mm,	Z =     0.344  mm,
	W =  -168.504 deg,	P =    -1.568 deg,	R =  -105.653 deg
};
P[1557]{
   GP1:
	UF : 7, UT : 3,	CONFIG : 'F U T, 0, 0, 0',
	X =  -294.443  mm,	Y =   168.806  mm,	Z =     0.500  mm,
	W =  -168.628 deg,	P =    -1.530 deg,	R =  -104.737 deg
};
P[1558]{
   GP1:
	UF : 7, UT : 3,	CONFIG : 'F U T, 0, 0, 0',
	X =  -300.389  mm,	Y =   158.022  mm,	Z =     0.821  mm,
	W =  -168.718 deg,	P =    -0.717 deg,	R =  -102.688 deg
};
P[1559]{
   GP1:
	UF : 7, UT : 3,	CONFIG : 'F U T, 0, 0, 0',
	X =  -308.417  mm,	Y =   141.685  mm,	Z =     0.916  mm,
	W =  -168.273 deg,	P =     0.590 deg,	R =   -99.646 deg
};
P[1560]{
   GP1:
	UF : 7, UT : 3,	CONFIG : 'F U T, 0, 0, 0',
	X =  -311.010  mm,	Y =   135.902  mm,	Z =     0.854  mm,
	W =  -168.139 deg,	P =     1.059 deg,	R =   -98.451 deg
};
P[1561]{
   GP1:
	UF : 7, UT : 3,	CONFIG : 'F U T, 0, 0, 0',
	X =  -315.265  mm,	Y =   125.737  mm,	Z =     0.576  mm,
	W =  -167.876 deg,	P =     2.240 deg,	R =   -96.686 deg
};
P[1562]{
   GP1:
	UF : 7, UT : 3,	CONFIG : 'F U T, 0, 0, 0',
	X =  -316.505  mm,	Y =   122.550  mm,	Z =     0.448  mm,
	W =  -167.781 deg,	P =     2.349 deg,	R =   -96.007 deg
};
P[1563]{
   GP1:
	UF : 7, UT : 3,	CONFIG : 'F U T, 0, 0, 0',
	X =  -317.757  mm,	Y =   119.272  mm,	Z =     0.316  mm,
	W =  -167.712 deg,	P =     2.253 deg,	R =   -95.560 deg
};
P[1564]{
   GP1:
	UF : 7, UT : 3,	CONFIG : 'F U T, 0, 0, 0',
	X =  -319.128  mm,	Y =   115.553  mm,	Z =     0.181  mm,
	W =  -167.649 deg,	P =     1.897 deg,	R =   -94.822 deg
};
P[1565]{
   GP1:
	UF : 7, UT : 3,	CONFIG : 'F U T, 0, 0, 0',
	X =  -321.857  mm,	Y =   107.699  mm,	Z =     0.000  mm,
	W =  -167.562 deg,	P =     0.788 deg,	R =   -92.833 deg
};
P[1566]{
   GP1:
	UF : 7, UT : 3,	CONFIG : 'F U T, 0, 0, 0',
	X =  -321.857  mm,	Y =   107.699  mm,	Z =     0.000  mm,
	W =  -167.562 deg,	P =     0.788 deg,	R =   -92.833 deg
};
P[1567]{
   GP1:
	UF : 7, UT : 3,	CONFIG : 'F U T, 0, 0, 0',
	X =  -321.857  mm,	Y =   107.699  mm,	Z =     0.000  mm,
	W =  -167.562 deg,	P =     0.788 deg,	R =   -92.833 deg
};
P[1568]{
   GP1:
	UF : 7, UT : 3,	CONFIG : 'F U T, 0, 0, 0',
	X =  -321.857  mm,	Y =   107.699  mm,	Z =     0.000  mm,
	W =  -167.562 deg,	P =     0.788 deg,	R =   -92.833 deg
};
P[1569]{
   GP1:
	UF : 7, UT : 3,	CONFIG : 'F U T, 0, 1, 0',
	X =  -336.714  mm,	Y =    42.617  mm,	Z =     0.000  mm,
	W =  -167.375 deg,	P =    -0.012 deg,	R =   -82.107 deg
};
P[1570]{
   GP1:
	UF : 7, UT : 3,	CONFIG : 'F U T, 0, 1, 0',
	X =  -336.714  mm,	Y =    42.617  mm,	Z =     0.000  mm,
	W =  -167.375 deg,	P =    -0.012 deg,	R =   -82.107 deg
};
P[1571]{
   GP1:
	UF : 7, UT : 3,	CONFIG : 'F U T, 0, 1, 0',
	X =  -336.714  mm,	Y =    42.617  mm,	Z =     0.000  mm,
	W =  -167.375 deg,	P =    -0.012 deg,	R =   -82.107 deg
};
P[1572]{
   GP1:
	UF : 7, UT : 3,	CONFIG : 'F U T, 0, 1, 0',
	X =  -336.714  mm,	Y =    42.617  mm,	Z =     0.000  mm,
	W =  -167.375 deg,	P =    -0.012 deg,	R =   -82.107 deg
};
P[1573]{
   GP1:
	UF : 7, UT : 3,	CONFIG : 'F U T, 0, 1, 0',
	X =  -338.645  mm,	Y =    22.718  mm,	Z =     0.002  mm,
	W =  -167.369 deg,	P =    -0.002 deg,	R =   -78.795 deg
};
P[1574]{
   GP1:
	UF : 7, UT : 3,	CONFIG : 'F U T, 0, 1, 0',
	X =  -339.418  mm,	Y =     0.000  mm,	Z =     0.000  mm,
	W =  -167.361 deg,	P =     0.008 deg,	R =   -75.587 deg
};
P[1575]{
   GP1:
	UF : 7, UT : 3,	CONFIG : 'F U T, 0, 1, 0',
	X =  -339.418  mm,	Y =     0.000  mm,	Z =     0.000  mm,
	W =  -167.361 deg,	P =     0.008 deg,	R =   -75.587 deg
};
P[1576]{
   GP1:
	UF : 7, UT : 3,	CONFIG : 'F U T, 0, 1, 0',
	X =  -339.418  mm,	Y =     0.000  mm,	Z =     0.000  mm,
	W =  -167.361 deg,	P =     0.008 deg,	R =   -75.587 deg
};
P[1577]{
   GP1:
	UF : 7, UT : 3,	CONFIG : 'F U T, 0, 1, 0',
	X =  -339.418  mm,	Y =     0.000  mm,	Z =     0.000  mm,
	W =  -167.361 deg,	P =     0.008 deg,	R =   -75.587 deg
};
P[1578]{
   GP1:
	UF : 7, UT : 3,	CONFIG : 'F U T, 0, 1, 0',
	X =  -336.284  mm,	Y =     0.000  mm,	Z =     0.000  mm,
	W =  -167.362 deg,	P =     0.007 deg,	R =   -75.584 deg
};
P[1579]{
   GP1:
	UF : 7, UT : 3,	CONFIG : 'F U T, 0, 1, 0',
	X =  -336.284  mm,	Y =     0.000  mm,	Z =     0.000  mm,
	W =  -167.362 deg,	P =     0.007 deg,	R =   -75.584 deg
};
P[1580]{
   GP1:
	UF : 7, UT : 3,	CONFIG : 'F U T, 0, 1, 0',
	X =  -336.284  mm,	Y =     0.000  mm,	Z =     0.000  mm,
	W =  -167.362 deg,	P =     0.007 deg,	R =   -75.584 deg
};
P[1581]{
   GP1:
	UF : 7, UT : 3,	CONFIG : 'F U T, 0, 1, 0',
	X =  -336.284  mm,	Y =     0.000  mm,	Z =     0.000  mm,
	W =  -167.362 deg,	P =     0.007 deg,	R =   -75.584 deg
};
P[1582]{
   GP1:
	UF : 7, UT : 3,	CONFIG : 'F U T, 0, 1, 0',
	X =  -335.525  mm,	Y =    22.441  mm,	Z =     0.002  mm,
	W =  -167.368 deg,	P =    -0.003 deg,	R =   -78.779 deg
};
P[1583]{
   GP1:
	UF : 7, UT : 3,	CONFIG : 'F U T, 0, 1, 0',
	X =  -333.802  mm,	Y =    40.612  mm,	Z =     0.000  mm,
	W =  -167.373 deg,	P =    -0.011 deg,	R =   -82.338 deg
};
P[1584]{
   GP1:
	UF : 7, UT : 3,	CONFIG : 'F U T, 0, 1, 0',
	X =  -333.802  mm,	Y =    40.612  mm,	Z =     0.000  mm,
	W =  -167.373 deg,	P =    -0.011 deg,	R =   -82.338 deg
};
P[1585]{
   GP1:
	UF : 7, UT : 3,	CONFIG : 'F U T, 0, 1, 0',
	X =  -333.802  mm,	Y =    40.612  mm,	Z =     0.000  mm,
	W =  -167.373 deg,	P =    -0.011 deg,	R =   -82.338 deg
};
P[1586]{
   GP1:
	UF : 7, UT : 3,	CONFIG : 'F U T, 0, 1, 0',
	X =  -333.802  mm,	Y =    40.612  mm,	Z =     0.000  mm,
	W =  -167.373 deg,	P =    -0.011 deg,	R =   -82.338 deg
};
P[1587]{
   GP1:
	UF : 7, UT : 3,	CONFIG : 'F U T, 0, 0, 0',
	X =  -318.375  mm,	Y =   108.240  mm,	Z =     0.000  mm,
	W =  -167.509 deg,	P =     0.852 deg,	R =   -93.749 deg
};
P[1588]{
   GP1:
	UF : 7, UT : 3,	CONFIG : 'F U T, 0, 0, 0',
	X =  -318.375  mm,	Y =   108.240  mm,	Z =     0.000  mm,
	W =  -167.509 deg,	P =     0.852 deg,	R =   -93.749 deg
};
P[1589]{
   GP1:
	UF : 7, UT : 3,	CONFIG : 'F U T, 0, 0, 0',
	X =  -318.375  mm,	Y =   108.240  mm,	Z =     0.000  mm,
	W =  -167.509 deg,	P =     0.852 deg,	R =   -93.749 deg
};
P[1590]{
   GP1:
	UF : 7, UT : 3,	CONFIG : 'F U T, 0, 0, 0',
	X =  -318.375  mm,	Y =   108.240  mm,	Z =     0.000  mm,
	W =  -167.509 deg,	P =     0.852 deg,	R =   -93.749 deg
};
P[1591]{
   GP1:
	UF : 7, UT : 3,	CONFIG : 'F U T, 0, 0, 0',
	X =  -316.026  mm,	Y =   114.910  mm,	Z =     0.154  mm,
	W =  -167.593 deg,	P =     1.801 deg,	R =   -94.835 deg
};
P[1592]{
   GP1:
	UF : 7, UT : 3,	CONFIG : 'F U T, 0, 0, 0',
	X =  -313.390  mm,	Y =   121.931  mm,	Z =     0.412  mm,
	W =  -167.792 deg,	P =     2.272 deg,	R =   -96.182 deg
};
P[1593]{
   GP1:
	UF : 7, UT : 3,	CONFIG : 'F U T, 0, 0, 0',
	X =  -312.127  mm,	Y =   125.119  mm,	Z =     0.537  mm,
	W =  -167.911 deg,	P =     2.182 deg,	R =   -96.819 deg
};
P[1594]{
   GP1:
	UF : 7, UT : 3,	CONFIG : 'F U T, 0, 0, 0',
	X =  -306.435  mm,	Y =   138.497  mm,	Z =     0.844  mm,
	W =  -168.299 deg,	P =     0.746 deg,	R =   -99.279 deg
};
P[1595]{
   GP1:
	UF : 7, UT : 3,	CONFIG : 'F U T, 0, 0, 0',
	X =  -298.063  mm,	Y =   155.695  mm,	Z =     0.777  mm,
	W =  -168.664 deg,	P =    -0.630 deg,	R =  -102.519 deg
};
P[1596]{
   GP1:
	UF : 7, UT : 3,	CONFIG : 'F U T, 0, 0, 0',
	X =  -291.601  mm,	Y =   167.464  mm,	Z =     0.447  mm,
	W =  -168.582 deg,	P =    -1.468 deg,	R =  -104.764 deg
};
P[1597]{
   GP1:
	UF : 7, UT : 3,	CONFIG : 'F U T, 0, 0, 0',
	X =  -286.518  mm,	Y =   176.040  mm,	Z =     0.148  mm,
	W =  -168.306 deg,	P =    -1.357 deg,	R =  -106.495 deg
};
P[1598]{
   GP1:
	UF : 7, UT : 3,	CONFIG : 'F U T, 0, 0, 0',
	X =  -283.127  mm,	Y =   181.427  mm,	Z =     0.000  mm,
	W =  -168.129 deg,	P =    -0.912 deg,	R =  -107.395 deg
};
P[1599]{
   GP1:
	UF : 7, UT : 3,	CONFIG : 'F U T, 0, 0, 0',
	X =  -283.127  mm,	Y =   181.427  mm,	Z =     0.000  mm,
	W =  -168.129 deg,	P =    -0.912 deg,	R =  -107.395 deg
};
P[1600]{
   GP1:
	UF : 7, UT : 3,	CONFIG : 'F U T, 0, 0, 0',
	X =  -283.127  mm,	Y =   181.427  mm,	Z =     0.000  mm,
	W =  -168.129 deg,	P =    -0.912 deg,	R =  -107.395 deg
};
P[1601]{
   GP1:
	UF : 7, UT : 3,	CONFIG : 'F U T, 0, 0, 0',
	X =  -283.127  mm,	Y =   181.427  mm,	Z =     0.000  mm,
	W =  -168.129 deg,	P =    -0.912 deg,	R =  -107.395 deg
};
P[1602]{
   GP1:
	UF : 7, UT : 3,	CONFIG : 'F U T, 0, 0, 0',
	X =  -239.888  mm,	Y =   235.660  mm,	Z =     0.000  mm,
	W =  -167.384 deg,	P =     0.111 deg,	R =  -119.940 deg
};
P[1603]{
   GP1:
	UF : 7, UT : 3,	CONFIG : 'F U T, 0, 0, 0',
	X =  -239.888  mm,	Y =   235.660  mm,	Z =     0.000  mm,
	W =  -167.384 deg,	P =     0.111 deg,	R =  -119.940 deg
};
P[1604]{
   GP1:
	UF : 7, UT : 3,	CONFIG : 'F U T, 0, 0, 0',
	X =  -239.888  mm,	Y =   235.660  mm,	Z =     0.000  mm,
	W =  -167.384 deg,	P =     0.111 deg,	R =  -119.940 deg
};
P[1605]{
   GP1:
	UF : 7, UT : 3,	CONFIG : 'F U T, 0, 0, 0',
	X =  -239.888  mm,	Y =   235.660  mm,	Z =     0.000  mm,
	W =  -167.384 deg,	P =     0.111 deg,	R =  -119.940 deg
};
P[1606]{
   GP1:
	UF : 7, UT : 3,	CONFIG : 'F U T, 0, 0, 0',
	X =  -228.981  mm,	Y =   246.264  mm,	Z =     0.017  mm,
	W =  -167.375 deg,	P =     0.046 deg,	R =  -122.062 deg
};
P[1607]{
   GP1:
	UF : 7, UT : 3,	CONFIG : 'F U T, 0, 0, 0',
	X =  -219.290  mm,	Y =   254.939  mm,	Z =     0.019  mm,
	W =  -167.363 deg,	P =    -0.008 deg,	R =  -124.222 deg
};
P[1608]{
   GP1:
	UF : 7, UT : 3,	CONFIG : 'F U T, 0, 0, 0',
	X =  -206.106  mm,	Y =   265.711  mm,	Z =     0.013  mm,
	W =  -167.366 deg,	P =    -0.009 deg,	R =  -127.181 deg
};
P[1609]{
   GP1:
	UF : 7, UT : 3,	CONFIG : 'F U T, 0, 0, 0',
	X =  -192.144  mm,	Y =   275.960  mm,	Z =     0.006  mm,
	W =  -167.369 deg,	P =    -0.009 deg,	R =  -130.086 deg
};
P[1610]{
   GP1:
	UF : 7, UT : 3,	CONFIG : 'F U T, 0, 0, 0',
	X =  -176.372  mm,	Y =   286.317  mm,	Z =     0.000  mm,
	W =  -167.372 deg,	P =    -0.010 deg,	R =  -132.837 deg
};
P[1611]{
   GP1:
	UF : 7, UT : 3,	CONFIG : 'F U T, 0, 0, 0',
	X =  -176.372  mm,	Y =   286.317  mm,	Z =     0.000  mm,
	W =  -167.372 deg,	P =    -0.010 deg,	R =  -132.837 deg
};
P[1612]{
   GP1:
	UF : 7, UT : 3,	CONFIG : 'F U T, 0, 0, 0',
	X =  -176.372  mm,	Y =   286.317  mm,	Z =     0.000  mm,
	W =  -167.372 deg,	P =    -0.010 deg,	R =  -132.837 deg
};
P[1613]{
   GP1:
	UF : 7, UT : 3,	CONFIG : 'F U T, 0, 0, 0',
	X =  -176.372  mm,	Y =   286.317  mm,	Z =     0.000  mm,
	W =  -167.372 deg,	P =    -0.010 deg,	R =  -132.837 deg
};
P[1614]{
   GP1:
	UF : 7, UT : 3,	CONFIG : 'F U T, 0, 0, 0',
	X =  -113.873  mm,	Y =   316.396  mm,	Z =     0.000  mm,
	W =  -167.364 deg,	P =     0.003 deg,	R =  -144.959 deg
};
P[1615]{
   GP1:
	UF : 7, UT : 3,	CONFIG : 'F U T, 0, 0, 0',
	X =  -113.873  mm,	Y =   316.396  mm,	Z =     0.000  mm,
	W =  -167.364 deg,	P =     0.003 deg,	R =  -144.959 deg
};
P[1616]{
   GP1:
	UF : 7, UT : 3,	CONFIG : 'F U T, 0, 0, 0',
	X =  -113.873  mm,	Y =   316.396  mm,	Z =     0.000  mm,
	W =  -167.364 deg,	P =     0.003 deg,	R =  -144.959 deg
};
P[1617]{
   GP1:
	UF : 7, UT : 3,	CONFIG : 'F U T, 0, 0, 0',
	X =  -113.873  mm,	Y =   316.396  mm,	Z =     0.000  mm,
	W =  -167.364 deg,	P =     0.003 deg,	R =  -144.959 deg
};
P[1618]{
   GP1:
	UF : 7, UT : 3,	CONFIG : 'F U T, 0, 0, 0',
	X =   -94.739  mm,	Y =   322.652  mm,	Z =     0.000  mm,
	W =  -167.364 deg,	P =     0.002 deg,	R =  -148.605 deg
};
P[1619]{
   GP1:
	UF : 7, UT : 3,	CONFIG : 'F U T, 0, 0, 0',
	X =   -74.506  mm,	Y =   327.916  mm,	Z =     0.000  mm,
	W =  -167.364 deg,	P =     0.001 deg,	R =  -152.122 deg
};
P[1620]{
   GP1:
	UF : 7, UT : 3,	CONFIG : 'F U T, 0, 0, 0',
	X =   -54.138  mm,	Y =   331.882  mm,	Z =     0.000  mm,
	W =  -167.364 deg,	P =     0.000 deg,	R =  -155.679 deg
};
P[1621]{
   GP1:
	UF : 7, UT : 3,	CONFIG : 'F U T, 0, 0, 0',
	X =   -34.683  mm,	Y =   334.472  mm,	Z =     0.000  mm,
	W =  -167.364 deg,	P =     0.000 deg,	R =  -159.479 deg
};
P[1622]{
   GP1:
	UF : 7, UT : 3,	CONFIG : 'F U T, 0, 0, 0',
	X =   -34.683  mm,	Y =   334.472  mm,	Z =     0.000  mm,
	W =  -167.364 deg,	P =     0.000 deg,	R =  -159.479 deg
};
P[1623]{
   GP1:
	UF : 7, UT : 3,	CONFIG : 'F U T, 0, 0, 0',
	X =   -34.683  mm,	Y =   334.472  mm,	Z =     0.000  mm,
	W =  -167.364 deg,	P =     0.000 deg,	R =  -159.479 deg
};
P[1624]{
   GP1:
	UF : 7, UT : 3,	CONFIG : 'F U T, 0, 0, 0',
	X =   -34.683  mm,	Y =   334.472  mm,	Z =     0.000  mm,
	W =  -167.364 deg,	P =     0.000 deg,	R =  -159.479 deg
};
P[1625]{
   GP1:
	UF : 7, UT : 3,	CONFIG : 'F U T, 0, 0, 0',
	X =    34.683  mm,	Y =   334.472  mm,	Z =     0.000  mm,
	W =  -167.363 deg,	P =     0.000 deg,	R =  -170.357 deg
};
P[1626]{
   GP1:
	UF : 7, UT : 3,	CONFIG : 'F U T, 0, 0, 0',
	X =    34.683  mm,	Y =   334.472  mm,	Z =     0.000  mm,
	W =  -167.363 deg,	P =     0.000 deg,	R =  -170.357 deg
};
P[1627]{
   GP1:
	UF : 7, UT : 3,	CONFIG : 'F U T, 0, 0, 0',
	X =    34.683  mm,	Y =   334.472  mm,	Z =     0.000  mm,
	W =  -167.363 deg,	P =     0.000 deg,	R =  -170.357 deg
};
P[1628]{
   GP1:
	UF : 7, UT : 3,	CONFIG : 'F U T, 0, 0, 0',
	X =    34.683  mm,	Y =   334.472  mm,	Z =     0.000  mm,
	W =  -167.363 deg,	P =     0.000 deg,	R =  -170.357 deg
};
P[1629]{
   GP1:
	UF : 7, UT : 3,	CONFIG : 'F U T, 0, 0, 0',
	X =    54.026  mm,	Y =   331.901  mm,	Z =     0.000  mm,
	W =  -167.364 deg,	P =     0.000 deg,	R =  -174.211 deg
};
P[1630]{
   GP1:
	UF : 7, UT : 3,	CONFIG : 'F U T, 0, 0, 0',
	X =    74.471  mm,	Y =   327.924  mm,	Z =     0.000  mm,
	W =  -167.364 deg,	P =     0.000 deg,	R =  -177.764 deg
};
P[1631]{
   GP1:
	UF : 7, UT : 3,	CONFIG : 'F U T, 0, 0, 0',
	X =    94.724  mm,	Y =   322.655  mm,	Z =     0.000  mm,
	W =  -167.364 deg,	P =     0.000 deg,	R =   178.709 deg
};
P[1632]{
   GP1:
	UF : 7, UT : 3,	CONFIG : 'F U T, 0, 0, 0',
	X =   113.873  mm,	Y =   316.396  mm,	Z =     0.000  mm,
	W =  -167.364 deg,	P =     0.000 deg,	R =   175.045 deg
};
P[1633]{
   GP1:
	UF : 7, UT : 3,	CONFIG : 'F U T, 0, 0, 0',
	X =   113.873  mm,	Y =   316.396  mm,	Z =     0.000  mm,
	W =  -167.364 deg,	P =     0.000 deg,	R =   175.045 deg
};
P[1634]{
   GP1:
	UF : 7, UT : 3,	CONFIG : 'F U T, 0, 0, 0',
	X =   113.873  mm,	Y =   316.396  mm,	Z =     0.000  mm,
	W =  -167.364 deg,	P =     0.000 deg,	R =   175.045 deg
};
P[1635]{
   GP1:
	UF : 7, UT : 3,	CONFIG : 'F U T, 0, 0, 0',
	X =   113.873  mm,	Y =   316.396  mm,	Z =     0.000  mm,
	W =  -167.364 deg,	P =     0.000 deg,	R =   175.045 deg
};
P[1636]{
   GP1:
	UF : 7, UT : 3,	CONFIG : 'F U T, 0, 0, 0',
	X =   176.372  mm,	Y =   286.317  mm,	Z =     0.000  mm,
	W =  -167.364 deg,	P =     0.001 deg,	R =   162.932 deg
};
P[1637]{
   GP1:
	UF : 7, UT : 3,	CONFIG : 'F U T, 0, 0, 0',
	X =   176.372  mm,	Y =   286.317  mm,	Z =     0.000  mm,
	W =  -167.364 deg,	P =     0.001 deg,	R =   162.932 deg
};
P[1638]{
   GP1:
	UF : 7, UT : 3,	CONFIG : 'F U T, 0, 0, 0',
	X =   176.372  mm,	Y =   286.317  mm,	Z =     0.000  mm,
	W =  -167.364 deg,	P =     0.001 deg,	R =   162.932 deg
};
P[1639]{
   GP1:
	UF : 7, UT : 3,	CONFIG : 'F U T, 0, 0, 0',
	X =   176.372  mm,	Y =   286.317  mm,	Z =     0.000  mm,
	W =  -167.364 deg,	P =     0.001 deg,	R =   162.932 deg
};
P[1640]{
   GP1:
	UF : 7, UT : 3,	CONFIG : 'F U T, 0, 0, 0',
	X =   194.026  mm,	Y =   274.652  mm,	Z =     0.000  mm,
	W =  -167.364 deg,	P =     0.000 deg,	R =   159.841 deg
};
P[1641]{
   GP1:
	UF : 7, UT : 3,	CONFIG : 'F U T, 0, 0, 0',
	X =   209.311  mm,	Y =   263.178  mm,	Z =     0.001  mm,
	W =  -167.364 deg,	P =     0.000 deg,	R =   156.548 deg
};
P[1642]{
   GP1:
	UF : 7, UT : 3,	CONFIG : 'F U T, 0, 0, 0',
	X =   224.067  mm,	Y =   250.758  mm,	Z =     0.001  mm,
	W =  -167.365 deg,	P =    -0.001 deg,	R =   153.280 deg
};
P[1643]{
   GP1:
	UF : 7, UT : 3,	CONFIG : 'F U T, 0, 0, 0',
	X =   239.888  mm,	Y =   235.660  mm,	Z =     0.000  mm,
	W =  -167.365 deg,	P =    -0.001 deg,	R =   150.048 deg
};
P[1644]{
   GP1:
	UF : 7, UT : 3,	CONFIG : 'F U T, 0, 0, 0',
	X =   239.888  mm,	Y =   235.660  mm,	Z =     0.000  mm,
	W =  -167.365 deg,	P =    -0.001 deg,	R =   150.048 deg
};
P[1645]{
   GP1:
	UF : 7, UT : 3,	CONFIG : 'F U T, 0, 0, 0',
	X =   239.888  mm,	Y =   235.660  mm,	Z =     0.000  mm,
	W =  -167.365 deg,	P =    -0.001 deg,	R =   150.048 deg
};
P[1646]{
   GP1:
	UF : 7, UT : 3,	CONFIG : 'F U T, 0, 0, 0',
	X =   239.888  mm,	Y =   235.660  mm,	Z =     0.000  mm,
	W =  -167.365 deg,	P =    -0.001 deg,	R =   150.048 deg
};
P[1647]{
   GP1:
	UF : 7, UT : 3,	CONFIG : 'F U T, 0, 0, 0',
	X =   283.127  mm,	Y =   181.427  mm,	Z =     0.000  mm,
	W =  -167.364 deg,	P =     0.002 deg,	R =   137.508 deg
};
P[1648]{
   GP1:
	UF : 7, UT : 3,	CONFIG : 'F U T, 0, 0, 0',
	X =   283.127  mm,	Y =   181.427  mm,	Z =     0.000  mm,
	W =  -167.364 deg,	P =     0.002 deg,	R =   137.508 deg
};
P[1649]{
   GP1:
	UF : 7, UT : 3,	CONFIG : 'F U T, 0, 0, 0',
	X =   283.127  mm,	Y =   181.427  mm,	Z =     0.000  mm,
	W =  -167.364 deg,	P =     0.002 deg,	R =   137.508 deg
};
P[1650]{
   GP1:
	UF : 7, UT : 3,	CONFIG : 'F U T, 0, 0, 0',
	X =   283.127  mm,	Y =   181.427  mm,	Z =     0.000  mm,
	W =  -167.364 deg,	P =     0.002 deg,	R =   137.508 deg
};
P[1651]{
   GP1:
	UF : 7, UT : 3,	CONFIG : 'F U T, 0, 0, 0',
	X =   293.822  mm,	Y =   163.545  mm,	Z =     0.000  mm,
	W =  -167.364 deg,	P =     0.001 deg,	R =   134.145 deg
};
P[1652]{
   GP1:
	UF : 7, UT : 3,	CONFIG : 'F U T, 0, 0, 0',
	X =   303.186  mm,	Y =   145.446  mm,	Z =     0.000  mm,
	W =  -167.364 deg,	P =     0.000 deg,	R =   130.742 deg
};
P[1653]{
   GP1:
	UF : 7, UT : 3,	CONFIG : 'F U T, 0, 0, 0',
	X =   311.314  mm,	Y =   127.116  mm,	Z =     0.000  mm,
	W =  -167.365 deg,	P =    -0.001 deg,	R =   127.286 deg
};
P[1654]{
   GP1:
	UF : 7, UT : 3,	CONFIG : 'F U T, 0, 0, 0',
	X =   318.375  mm,	Y =   108.240  mm,	Z =     0.000  mm,
	W =  -167.365 deg,	P =    -0.002 deg,	R =   123.856 deg
};
P[1655]{
   GP1:
	UF : 7, UT : 3,	CONFIG : 'F U T, 0, 0, 0',
	X =   318.375  mm,	Y =   108.240  mm,	Z =     0.000  mm,
	W =  -167.365 deg,	P =    -0.002 deg,	R =   123.856 deg
};
P[1656]{
   GP1:
	UF : 7, UT : 3,	CONFIG : 'F U T, 0, 0, 0',
	X =   318.375  mm,	Y =   108.240  mm,	Z =     0.000  mm,
	W =  -167.365 deg,	P =    -0.002 deg,	R =   123.856 deg
};
P[1657]{
   GP1:
	UF : 7, UT : 3,	CONFIG : 'F U T, 0, 0, 0',
	X =   318.375  mm,	Y =   108.240  mm,	Z =     0.000  mm,
	W =  -167.365 deg,	P =    -0.002 deg,	R =   123.856 deg
};
P[1658]{
   GP1:
	UF : 7, UT : 3,	CONFIG : 'F U T, 0, 0, 0',
	X =   333.802  mm,	Y =    40.612  mm,	Z =     0.000  mm,
	W =  -167.364 deg,	P =     0.001 deg,	R =   112.508 deg
};
P[1659]{
   GP1:
	UF : 7, UT : 3,	CONFIG : 'F U T, 0, 0, 0',
	X =   333.802  mm,	Y =    40.612  mm,	Z =     0.000  mm,
	W =  -167.364 deg,	P =     0.001 deg,	R =   112.508 deg
};
P[1660]{
   GP1:
	UF : 7, UT : 3,	CONFIG : 'F U T, 0, 0, 0',
	X =   333.802  mm,	Y =    40.612  mm,	Z =     0.000  mm,
	W =  -167.364 deg,	P =     0.001 deg,	R =   112.508 deg
};
P[1661]{
   GP1:
	UF : 7, UT : 3,	CONFIG : 'F U T, 0, 0, 0',
	X =   333.802  mm,	Y =    40.612  mm,	Z =     0.000  mm,
	W =  -167.364 deg,	P =     0.001 deg,	R =   112.508 deg
};
P[1662]{
   GP1:
	UF : 7, UT : 3,	CONFIG : 'F U T, 0, 0, 0',
	X =   335.518  mm,	Y =    22.564  mm,	Z =     0.000  mm,
	W =  -167.364 deg,	P =     0.000 deg,	R =   108.910 deg
};
P[1663]{
   GP1:
	UF : 7, UT : 3,	CONFIG : 'F U T, 0, 0, 0',
	X =   336.284  mm,	Y =     0.000  mm,	Z =     0.000  mm,
	W =  -167.364 deg,	P =    -0.001 deg,	R =   105.689 deg
};
P[1664]{
   GP1:
	UF : 7, UT : 3,	CONFIG : 'F U T, 0, 0, 0',
	X =   336.284  mm,	Y =     0.000  mm,	Z =     0.000  mm,
	W =  -167.364 deg,	P =    -0.001 deg,	R =   105.689 deg
};
P[1665]{
   GP1:
	UF : 7, UT : 3,	CONFIG : 'F U T, 0, 0, 0',
	X =   336.284  mm,	Y =     0.000  mm,	Z =     0.000  mm,
	W =  -167.364 deg,	P =    -0.001 deg,	R =   105.689 deg
};
P[1666]{
   GP1:
	UF : 7, UT : 3,	CONFIG : 'F U T, 0, 0, 0',
	X =   336.284  mm,	Y =     0.000  mm,	Z =     0.000  mm,
	W =  -167.364 deg,	P =    -0.001 deg,	R =   105.689 deg
};
P[1667]{
   GP1:
	UF : 7, UT : 3,	CONFIG : 'F U T, 0, 0, 0',
	X =   333.150  mm,	Y =     0.000  mm,	Z =     0.000  mm,
	W =  -167.364 deg,	P =    -0.001 deg,	R =   105.691 deg
};
P[1668]{
   GP1:
	UF : 7, UT : 3,	CONFIG : 'F U T, 0, 0, 0',
	X =   333.150  mm,	Y =     0.000  mm,	Z =     0.000  mm,
	W =  -167.364 deg,	P =    -0.001 deg,	R =   105.691 deg
};
P[1669]{
   GP1:
	UF : 7, UT : 3,	CONFIG : 'F U T, 0, 0, 0',
	X =   333.150  mm,	Y =     0.000  mm,	Z =     0.000  mm,
	W =  -167.364 deg,	P =    -0.001 deg,	R =   105.691 deg
};
P[1670]{
   GP1:
	UF : 7, UT : 3,	CONFIG : 'F U T, 0, 0, 0',
	X =   333.150  mm,	Y =     0.000  mm,	Z =     0.000  mm,
	W =  -167.364 deg,	P =    -0.001 deg,	R =   105.691 deg
};
P[1671]{
   GP1:
	UF : 7, UT : 3,	CONFIG : 'F U T, 0, 0, 0',
	X =   332.435  mm,	Y =    21.735  mm,	Z =     0.000  mm,
	W =  -167.364 deg,	P =     0.000 deg,	R =   108.776 deg
};
P[1672]{
   GP1:
	UF : 7, UT : 3,	CONFIG : 'F U T, 0, 0, 0',
	X =   330.845  mm,	Y =    38.971  mm,	Z =     0.000  mm,
	W =  -167.364 deg,	P =     0.001 deg,	R =   112.270 deg
};
P[1673]{
   GP1:
	UF : 7, UT : 3,	CONFIG : 'F U T, 0, 0, 0',
	X =   330.845  mm,	Y =    38.971  mm,	Z =     0.000  mm,
	W =  -167.364 deg,	P =     0.001 deg,	R =   112.270 deg
};
P[1674]{
   GP1:
	UF : 7, UT : 3,	CONFIG : 'F U T, 0, 0, 0',
	X =   330.845  mm,	Y =    38.971  mm,	Z =     0.000  mm,
	W =  -167.364 deg,	P =     0.001 deg,	R =   112.270 deg
};
P[1675]{
   GP1:
	UF : 7, UT : 3,	CONFIG : 'F U T, 0, 0, 0',
	X =   330.845  mm,	Y =    38.971  mm,	Z =     0.000  mm,
	W =  -167.364 deg,	P =     0.001 deg,	R =   112.270 deg
};
P[1676]{
   GP1:
	UF : 7, UT : 3,	CONFIG : 'F U T, 0, 0, 0',
	X =   315.007  mm,	Y =   108.436  mm,	Z =     0.000  mm,
	W =  -167.365 deg,	P =    -0.002 deg,	R =   124.625 deg
};
P[1677]{
   GP1:
	UF : 7, UT : 3,	CONFIG : 'F U T, 0, 0, 0',
	X =   315.007  mm,	Y =   108.436  mm,	Z =     0.000  mm,
	W =  -167.365 deg,	P =    -0.002 deg,	R =   124.625 deg
};
P[1678]{
   GP1:
	UF : 7, UT : 3,	CONFIG : 'F U T, 0, 0, 0',
	X =   315.007  mm,	Y =   108.436  mm,	Z =     0.000  mm,
	W =  -167.365 deg,	P =    -0.002 deg,	R =   124.625 deg
};
P[1679]{
   GP1:
	UF : 7, UT : 3,	CONFIG : 'F U T, 0, 0, 0',
	X =   315.007  mm,	Y =   108.436  mm,	Z =     0.000  mm,
	W =  -167.365 deg,	P =    -0.002 deg,	R =   124.625 deg
};
P[1680]{
   GP1:
	UF : 7, UT : 3,	CONFIG : 'F U T, 0, 0, 0',
	X =   307.327  mm,	Y =   128.571  mm,	Z =     0.000  mm,
	W =  -167.365 deg,	P =    -0.001 deg,	R =   127.726 deg
};
P[1681]{
   GP1:
	UF : 7, UT : 3,	CONFIG : 'F U T, 0, 0, 0',
	X =   299.459  mm,	Y =   145.950  mm,	Z =     0.000  mm,
	W =  -167.364 deg,	P =     0.000 deg,	R =   131.022 deg
};
P[1682]{
   GP1:
	UF : 7, UT : 3,	CONFIG : 'F U T, 0, 0, 0',
	X =   290.635  mm,	Y =   162.830  mm,	Z =     0.000  mm,
	W =  -167.364 deg,	P =     0.001 deg,	R =   134.337 deg
};
P[1683]{
   GP1:
	UF : 7, UT : 3,	CONFIG : 'F U T, 0, 0, 0',
	X =   281.171  mm,	Y =   178.658  mm,	Z =     0.000  mm,
	W =  -167.364 deg,	P =     0.002 deg,	R =   137.765 deg
};
P[1684]{
   GP1:
	UF : 7, UT : 3,	CONFIG : 'F U T, 0, 0, 0',
	X =   281.171  mm,	Y =   178.658  mm,	Z =     0.000  mm,
	W =  -167.364 deg,	P =     0.002 deg,	R =   137.765 deg
};
P[1685]{
   GP1:
	UF : 7, UT : 3,	CONFIG : 'F U T, 0, 0, 0',
	X =   281.171  mm,	Y =   178.658  mm,	Z =     0.000  mm,
	W =  -167.364 deg,	P =     0.002 deg,	R =   137.765 deg
};
P[1686]{
   GP1:
	UF : 7, UT : 3,	CONFIG : 'F U T, 0, 0, 0',
	X =   281.171  mm,	Y =   178.658  mm,	Z =     0.000  mm,
	W =  -167.364 deg,	P =     0.002 deg,	R =   137.765 deg
};
P[1687]{
   GP1:
	UF : 7, UT : 3,	CONFIG : 'F U T, 0, 0, 0',
	X =   236.748  mm,	Y =   234.368  mm,	Z =     0.000  mm,
	W =  -167.365 deg,	P =    -0.002 deg,	R =   149.949 deg
};
P[1688]{
   GP1:
	UF : 7, UT : 3,	CONFIG : 'F U T, 0, 0, 0',
	X =   236.748  mm,	Y =   234.368  mm,	Z =     0.000  mm,
	W =  -167.365 deg,	P =    -0.002 deg,	R =   149.949 deg
};
P[1689]{
   GP1:
	UF : 7, UT : 3,	CONFIG : 'F U T, 0, 0, 0',
	X =   236.748  mm,	Y =   234.368  mm,	Z =     0.000  mm,
	W =  -167.365 deg,	P =    -0.002 deg,	R =   149.949 deg
};
P[1690]{
   GP1:
	UF : 7, UT : 3,	CONFIG : 'F U T, 0, 0, 0',
	X =   236.748  mm,	Y =   234.368  mm,	Z =     0.000  mm,
	W =  -167.365 deg,	P =    -0.002 deg,	R =   149.949 deg
};
P[1691]{
   GP1:
	UF : 7, UT : 3,	CONFIG : 'F U T, 0, 0, 0',
	X =   222.462  mm,	Y =   247.982  mm,	Z =     0.001  mm,
	W =  -167.364 deg,	P =    -0.001 deg,	R =   153.112 deg
};
P[1692]{
   GP1:
	UF : 7, UT : 3,	CONFIG : 'F U T, 0, 0, 0',
	X =   208.284  mm,	Y =   259.988  mm,	Z =     0.001  mm,
	W =  -167.364 deg,	P =     0.000 deg,	R =   156.369 deg
};
P[1693]{
   GP1:
	UF : 7, UT : 3,	CONFIG : 'F U T, 0, 0, 0',
	X =   193.321  mm,	Y =   271.319  mm,	Z =     0.000  mm,
	W =  -167.364 deg,	P =     0.001 deg,	R =   159.589 deg
};
P[1694]{
   GP1:
	UF : 7, UT : 3,	CONFIG : 'F U T, 0, 0, 0',
	X =   175.812  mm,	Y =   282.971  mm,	Z =     0.000  mm,
	W =  -167.364 deg,	P =     0.001 deg,	R =   162.742 deg
};
P[1695]{
   GP1:
	UF : 7, UT : 3,	CONFIG : 'F U T, 0, 0, 0',
	X =   175.812  mm,	Y =   282.971  mm,	Z =     0.000  mm,
	W =  -167.364 deg,	P =     0.001 deg,	R =   162.742 deg
};
P[1696]{
   GP1:
	UF : 7, UT : 3,	CONFIG : 'F U T, 0, 0, 0',
	X =   175.812  mm,	Y =   282.971  mm,	Z =     0.000  mm,
	W =  -167.364 deg,	P =     0.001 deg,	R =   162.742 deg
};
P[1697]{
   GP1:
	UF : 7, UT : 3,	CONFIG : 'F U T, 0, 0, 0',
	X =   175.812  mm,	Y =   282.971  mm,	Z =     0.000  mm,
	W =  -167.364 deg,	P =     0.001 deg,	R =   162.742 deg
};
P[1698]{
   GP1:
	UF : 7, UT : 3,	CONFIG : 'F U T, 0, 0, 0',
	X =   111.612  mm,	Y =   313.876  mm,	Z =     0.000  mm,
	W =  -167.364 deg,	P =     0.000 deg,	R =   174.997 deg
};
P[1699]{
   GP1:
	UF : 7, UT : 3,	CONFIG : 'F U T, 0, 0, 0',
	X =   111.612  mm,	Y =   313.876  mm,	Z =     0.000  mm,
	W =  -167.364 deg,	P =     0.000 deg,	R =   174.997 deg
};
P[1700]{
   GP1:
	UF : 7, UT : 3,	CONFIG : 'F U T, 0, 0, 0',
	X =   111.612  mm,	Y =   313.876  mm,	Z =     0.000  mm,
	W =  -167.364 deg,	P =     0.000 deg,	R =   174.997 deg
};
P[1701]{
   GP1:
	UF : 7, UT : 3,	CONFIG : 'F U T, 0, 0, 0',
	X =   111.612  mm,	Y =   313.876  mm,	Z =     0.000  mm,
	W =  -167.364 deg,	P =     0.000 deg,	R =   174.997 deg
};
P[1702]{
   GP1:
	UF : 7, UT : 3,	CONFIG : 'F U T, 0, 0, 0',
	X =    93.943  mm,	Y =   319.625  mm,	Z =     0.000  mm,
	W =  -167.364 deg,	P =     0.000 deg,	R =   178.691 deg
};
P[1703]{
   GP1:
	UF : 7, UT : 3,	CONFIG : 'F U T, 0, 0, 0',
	X =    74.624  mm,	Y =   324.672  mm,	Z =     0.000  mm,
	W =  -167.364 deg,	P =     0.000 deg,	R =  -177.914 deg
};
P[1704]{
   GP1:
	UF : 7, UT : 3,	CONFIG : 'F U T, 0, 0, 0',
	X =    55.260  mm,	Y =   328.516  mm,	Z =     0.000  mm,
	W =  -167.364 deg,	P =     0.000 deg,	R =  -174.482 deg
};
P[1705]{
   GP1:
	UF : 7, UT : 3,	CONFIG : 'F U T, 0, 0, 0',
	X =    35.625  mm,	Y =   331.228  mm,	Z =     0.000  mm,
	W =  -167.363 deg,	P =     0.000 deg,	R =  -171.083 deg
};
P[1706]{
   GP1:
	UF : 7, UT : 3,	CONFIG : 'F U T, 0, 0, 0',
	X =    35.625  mm,	Y =   331.228  mm,	Z =     0.000  mm,
	W =  -167.363 deg,	P =     0.000 deg,	R =  -171.083 deg
};
P[1707]{
   GP1:
	UF : 7, UT : 3,	CONFIG : 'F U T, 0, 0, 0',
	X =    35.625  mm,	Y =   331.228  mm,	Z =     0.000  mm,
	W =  -167.363 deg,	P =     0.000 deg,	R =  -171.083 deg
};
P[1708]{
   GP1:
	UF : 7, UT : 3,	CONFIG : 'F U T, 0, 0, 0',
	X =    35.625  mm,	Y =   331.228  mm,	Z =     0.000  mm,
	W =  -167.363 deg,	P =     0.000 deg,	R =  -171.083 deg
};
P[1709]{
   GP1:
	UF : 7, UT : 3,	CONFIG : 'F U T, 0, 0, 0',
	X =   -35.625  mm,	Y =   331.228  mm,	Z =     0.000  mm,
	W =  -167.364 deg,	P =     0.000 deg,	R =  -158.706 deg
};
P[1710]{
   GP1:
	UF : 7, UT : 3,	CONFIG : 'F U T, 0, 0, 0',
	X =   -35.625  mm,	Y =   331.228  mm,	Z =     0.000  mm,
	W =  -167.364 deg,	P =     0.000 deg,	R =  -158.706 deg
};
P[1711]{
   GP1:
	UF : 7, UT : 3,	CONFIG : 'F U T, 0, 0, 0',
	X =   -35.625  mm,	Y =   331.228  mm,	Z =     0.000  mm,
	W =  -167.364 deg,	P =     0.000 deg,	R =  -158.706 deg
};
P[1712]{
   GP1:
	UF : 7, UT : 3,	CONFIG : 'F U T, 0, 0, 0',
	X =   -35.625  mm,	Y =   331.228  mm,	Z =     0.000  mm,
	W =  -167.364 deg,	P =     0.000 deg,	R =  -158.706 deg
};
P[1713]{
   GP1:
	UF : 7, UT : 3,	CONFIG : 'F U T, 0, 0, 0',
	X =   -55.594  mm,	Y =   328.460  mm,	Z =     0.000  mm,
	W =  -167.364 deg,	P =     0.000 deg,	R =  -155.377 deg
};
P[1714]{
   GP1:
	UF : 7, UT : 3,	CONFIG : 'F U T, 0, 0, 0',
	X =   -74.863  mm,	Y =   324.616  mm,	Z =     0.000  mm,
	W =  -167.364 deg,	P =     0.001 deg,	R =  -151.954 deg
};
P[1715]{
   GP1:
	UF : 7, UT : 3,	CONFIG : 'F U T, 0, 0, 0',
	X =   -94.063  mm,	Y =   319.587  mm,	Z =     0.000  mm,
	W =  -167.364 deg,	P =     0.002 deg,	R =  -148.554 deg
};
P[1716]{
   GP1:
	UF : 7, UT : 3,	CONFIG : 'F U T, 0, 0, 0',
	X =  -111.612  mm,	Y =   313.876  mm,	Z =     0.000  mm,
	W =  -167.364 deg,	P =     0.003 deg,	R =  -144.856 deg
};
P[1717]{
   GP1:
	UF : 7, UT : 3,	CONFIG : 'F U T, 0, 0, 0',
	X =  -111.612  mm,	Y =   313.876  mm,	Z =     0.000  mm,
	W =  -167.364 deg,	P =     0.003 deg,	R =  -144.856 deg
};
P[1718]{
   GP1:
	UF : 7, UT : 3,	CONFIG : 'F U T, 0, 0, 0',
	X =  -111.612  mm,	Y =   313.876  mm,	Z =     0.000  mm,
	W =  -167.364 deg,	P =     0.003 deg,	R =  -144.856 deg
};
P[1719]{
   GP1:
	UF : 7, UT : 3,	CONFIG : 'F U T, 0, 0, 0',
	X =  -111.612  mm,	Y =   313.876  mm,	Z =     0.000  mm,
	W =  -167.364 deg,	P =     0.003 deg,	R =  -144.856 deg
};
P[1720]{
   GP1:
	UF : 7, UT : 3,	CONFIG : 'F U T, 0, 0, 0',
	X =  -175.812  mm,	Y =   282.971  mm,	Z =     0.000  mm,
	W =  -167.372 deg,	P =    -0.012 deg,	R =  -132.630 deg
};
P[1721]{
   GP1:
	UF : 7, UT : 3,	CONFIG : 'F U T, 0, 0, 0',
	X =  -175.812  mm,	Y =   282.971  mm,	Z =     0.000  mm,
	W =  -167.372 deg,	P =    -0.012 deg,	R =  -132.630 deg
};
P[1722]{
   GP1:
	UF : 7, UT : 3,	CONFIG : 'F U T, 0, 0, 0',
	X =  -175.812  mm,	Y =   282.971  mm,	Z =     0.000  mm,
	W =  -167.372 deg,	P =    -0.012 deg,	R =  -132.630 deg
};
P[1723]{
   GP1:
	UF : 7, UT : 3,	CONFIG : 'F U T, 0, 0, 0',
	X =  -175.812  mm,	Y =   282.971  mm,	Z =     0.000  mm,
	W =  -167.372 deg,	P =    -0.012 deg,	R =  -132.630 deg
};
P[1724]{
   GP1:
	UF : 7, UT : 3,	CONFIG : 'F U T, 0, 0, 0',
	X =  -191.133  mm,	Y =   272.844  mm,	Z =     0.006  mm,
	W =  -167.368 deg,	P =    -0.011 deg,	R =  -129.982 deg
};
P[1725]{
   GP1:
	UF : 7, UT : 3,	CONFIG : 'F U T, 0, 0, 0',
	X =  -203.884  mm,	Y =   263.459  mm,	Z =     0.013  mm,
	W =  -167.364 deg,	P =    -0.011 deg,	R =  -127.261 deg
};
P[1726]{
   GP1:
	UF : 7, UT : 3,	CONFIG : 'F U T, 0, 0, 0',
	X =  -216.129  mm,	Y =   253.518  mm,	Z =     0.019  mm,
	W =  -167.360 deg,	P =    -0.011 deg,	R =  -124.524 deg
};
P[1727]{
   GP1:
	UF : 7, UT : 3,	CONFIG : 'F U T, 0, 0, 0',
	X =  -226.532  mm,	Y =   244.258  mm,	Z =     0.017  mm,
	W =  -167.369 deg,	P =     0.050 deg,	R =  -122.162 deg
};
P[1728]{
   GP1:
	UF : 7, UT : 3,	CONFIG : 'F U T, 0, 0, 0',
	X =  -236.748  mm,	Y =   234.368  mm,	Z =     0.000  mm,
	W =  -167.373 deg,	P =     0.112 deg,	R =  -119.824 deg
};
P[1729]{
   GP1:
	UF : 7, UT : 3,	CONFIG : 'F U T, 0, 0, 0',
	X =  -236.748  mm,	Y =   234.368  mm,	Z =     0.000  mm,
	W =  -167.373 deg,	P =     0.112 deg,	R =  -119.824 deg
};
P[1730]{
   GP1:
	UF : 7, UT : 3,	CONFIG : 'F U T, 0, 0, 0',
	X =  -236.748  mm,	Y =   234.368  mm,	Z =     0.000  mm,
	W =  -167.373 deg,	P =     0.112 deg,	R =  -119.824 deg
};
P[1731]{
   GP1:
	UF : 7, UT : 3,	CONFIG : 'F U T, 0, 0, 0',
	X =  -236.748  mm,	Y =   234.368  mm,	Z =     0.000  mm,
	W =  -167.373 deg,	P =     0.112 deg,	R =  -119.824 deg
};
P[1732]{
   GP1:
	UF : 7, UT : 3,	CONFIG : 'F U T, 0, 0, 0',
	X =  -281.171  mm,	Y =   178.658  mm,	Z =     0.000  mm,
	W =  -168.073 deg,	P =    -1.033 deg,	R =  -107.631 deg
};
P[1733]{
   GP1:
	UF : 7, UT : 3,	CONFIG : 'F U T, 0, 0, 0',
	X =  -281.171  mm,	Y =   178.658  mm,	Z =     0.000  mm,
	W =  -168.073 deg,	P =    -1.033 deg,	R =  -107.631 deg
};
P[1734]{
   GP1:
	UF : 7, UT : 3,	CONFIG : 'F U T, 0, 0, 0',
	X =  -281.171  mm,	Y =   178.658  mm,	Z =     0.000  mm,
	W =  -168.073 deg,	P =    -1.033 deg,	R =  -107.631 deg
};
P[1735]{
   GP1:
	UF : 7, UT : 3,	CONFIG : 'F U T, 0, 0, 0',
	X =  -281.171  mm,	Y =   178.658  mm,	Z =     0.000  mm,
	W =  -168.073 deg,	P =    -1.033 deg,	R =  -107.631 deg
};
P[1736]{
   GP1:
	UF : 7, UT : 3,	CONFIG : 'F U T, 0, 0, 0',
	X =  -286.553  mm,	Y =   169.906  mm,	Z =     0.268  mm,
	W =  -168.381 deg,	P =    -1.470 deg,	R =  -105.670 deg
};
P[1737]{
   GP1:
	UF : 7, UT : 3,	CONFIG : 'F U T, 0, 0, 0',
	X =  -291.938  mm,	Y =   160.474  mm,	Z =     0.573  mm,
	W =  -168.622 deg,	P =    -1.101 deg,	R =  -103.675 deg
};
P[1738]{
   GP1:
	UF : 7, UT : 3,	CONFIG : 'F U T, 0, 0, 0',
	X =  -299.700  mm,	Y =   145.466  mm,	Z =     0.808  mm,
	W =  -168.486 deg,	P =     0.157 deg,	R =  -100.857 deg
};
P[1739]{
   GP1:
	UF : 7, UT : 3,	CONFIG : 'F U T, 0, 0, 0',
	X =  -305.945  mm,	Y =   131.825  mm,	Z =     0.706  mm,
	W =  -168.207 deg,	P =     1.310 deg,	R =   -98.236 deg
};
P[1740]{
   GP1:
	UF : 7, UT : 3,	CONFIG : 'F U T, 0, 0, 0',
	X =  -309.168  mm,	Y =   124.080  mm,	Z =     0.481  mm,
	W =  -167.904 deg,	P =     2.107 deg,	R =   -96.857 deg
};
P[1741]{
   GP1:
	UF : 7, UT : 3,	CONFIG : 'F U T, 0, 0, 0',
	X =  -311.646  mm,	Y =   117.710  mm,	Z =     0.245  mm,
	W =  -167.632 deg,	P =     2.022 deg,	R =   -95.617 deg
};
P[1742]{
   GP1:
	UF : 7, UT : 3,	CONFIG : 'F U T, 0, 0, 0',
	X =  -315.007  mm,	Y =   108.436  mm,	Z =     0.000  mm,
	W =  -167.446 deg,	P =     0.873 deg,	R =   -94.516 deg
};
P[1743]{
   GP1:
	UF : 7, UT : 3,	CONFIG : 'F U T, 0, 0, 0',
	X =  -315.007  mm,	Y =   108.436  mm,	Z =     0.000  mm,
	W =  -167.446 deg,	P =     0.873 deg,	R =   -94.516 deg
};
P[1744]{
   GP1:
	UF : 7, UT : 3,	CONFIG : 'F U T, 0, 0, 0',
	X =  -315.007  mm,	Y =   108.436  mm,	Z =     0.000  mm,
	W =  -167.446 deg,	P =     0.873 deg,	R =   -94.516 deg
};
P[1745]{
   GP1:
	UF : 7, UT : 3,	CONFIG : 'F U T, 0, 0, 0',
	X =  -315.007  mm,	Y =   108.436  mm,	Z =     0.000  mm,
	W =  -167.446 deg,	P =     0.873 deg,	R =   -94.516 deg
};
P[1746]{
   GP1:
	UF : 7, UT : 3,	CONFIG : 'F U T, 0, 1, 0',
	X =  -330.845  mm,	Y =    38.971  mm,	Z =     0.000  mm,
	W =  -167.371 deg,	P =    -0.011 deg,	R =   -82.160 deg
};
P[1747]{
   GP1:
	UF : 7, UT : 3,	CONFIG : 'F U T, 0, 1, 0',
	X =  -330.845  mm,	Y =    38.971  mm,	Z =     0.000  mm,
	W =  -167.371 deg,	P =    -0.011 deg,	R =   -82.160 deg
};
P[1748]{
   GP1:
	UF : 7, UT : 3,	CONFIG : 'F U T, 0, 1, 0',
	X =  -330.845  mm,	Y =    38.971  mm,	Z =     0.000  mm,
	W =  -167.371 deg,	P =    -0.011 deg,	R =   -82.160 deg
};
P[1749]{
   GP1:
	UF : 7, UT : 3,	CONFIG : 'F U T, 0, 1, 0',
	X =  -330.845  mm,	Y =    38.971  mm,	Z =     0.000  mm,
	W =  -167.371 deg,	P =    -0.011 deg,	R =   -82.160 deg
};
P[1750]{
   GP1:
	UF : 7, UT : 3,	CONFIG : 'F U T, 0, 1, 0',
	X =  -332.434  mm,	Y =    21.718  mm,	Z =     0.002  mm,
	W =  -167.367 deg,	P =    -0.003 deg,	R =   -78.671 deg
};
P[1751]{
   GP1:
	UF : 7, UT : 3,	CONFIG : 'F U T, 0, 1, 0',
	X =  -333.150  mm,	Y =     0.000  mm,	Z =     0.000  mm,
	W =  -167.362 deg,	P =     0.007 deg,	R =   -75.582 deg
};
P[1752]{
   GP1:
	UF : 7, UT : 3,	CONFIG : 'F U T, 0, 1, 0',
	X =  -333.150  mm,	Y =     0.000  mm,	Z =     0.000  mm,
	W =  -167.362 deg,	P =     0.007 deg,	R =   -75.582 deg
};
P[1753]{
   GP1:
	UF : 7, UT : 3,	CONFIG : 'F U T, 0, 1, 0',
	X =  -333.150  mm,	Y =     0.000  mm,	Z =     0.000  mm,
	W =  -167.362 deg,	P =     0.007 deg,	R =   -75.582 deg
};
P[1754]{
   GP1:
	UF : 7, UT : 3,	CONFIG : 'F U T, 0, 1, 0',
	X =  -333.150  mm,	Y =     0.000  mm,	Z =     0.000  mm,
	W =  -167.362 deg,	P =     0.007 deg,	R =   -75.582 deg
};
P[1755]{
   GP1:
	UF : 7, UT : 3,	CONFIG : 'F U T, 0, 1, 0',
	X =  -330.015  mm,	Y =     0.000  mm,	Z =     0.000  mm,
	W =  -167.362 deg,	P =     0.007 deg,	R =   -75.584 deg
};
P[1756]{
   GP1:
	UF : 7, UT : 3,	CONFIG : 'F U T, 0, 1, 0',
	X =  -330.015  mm,	Y =     0.000  mm,	Z =     0.000  mm,
	W =  -167.362 deg,	P =     0.007 deg,	R =   -75.584 deg
};
P[1757]{
   GP1:
	UF : 7, UT : 3,	CONFIG : 'F U T, 0, 1, 0',
	X =  -330.015  mm,	Y =     0.000  mm,	Z =     0.000  mm,
	W =  -167.362 deg,	P =     0.007 deg,	R =   -75.584 deg
};
P[1758]{
   GP1:
	UF : 7, UT : 3,	CONFIG : 'F U T, 0, 1, 0',
	X =  -330.015  mm,	Y =     0.000  mm,	Z =     0.000  mm,
	W =  -167.362 deg,	P =     0.007 deg,	R =   -75.584 deg
};
P[1759]{
   GP1:
	UF : 7, UT : 3,	CONFIG : 'F U T, 0, 1, 0',
	X =  -329.378  mm,	Y =    20.313  mm,	Z =     0.001  mm,
	W =  -167.367 deg,	P =    -0.003 deg,	R =   -78.441 deg
};
P[1760]{
   GP1:
	UF : 7, UT : 3,	CONFIG : 'F U T, 0, 1, 0',
	X =  -327.850  mm,	Y =    37.642  mm,	Z =     0.000  mm,
	W =  -167.370 deg,	P =    -0.011 deg,	R =   -81.388 deg
};
P[1761]{
   GP1:
	UF : 7, UT : 3,	CONFIG : 'F U T, 0, 1, 0',
	X =  -327.850  mm,	Y =    37.642  mm,	Z =     0.000  mm,
	W =  -167.370 deg,	P =    -0.011 deg,	R =   -81.388 deg
};
P[1762]{
   GP1:
	UF : 7, UT : 3,	CONFIG : 'F U T, 0, 1, 0',
	X =  -327.850  mm,	Y =    37.642  mm,	Z =     0.000  mm,
	W =  -167.370 deg,	P =    -0.011 deg,	R =   -81.388 deg
};
P[1763]{
   GP1:
	UF : 7, UT : 3,	CONFIG : 'F U T, 0, 1, 0',
	X =  -327.850  mm,	Y =    37.642  mm,	Z =     0.000  mm,
	W =  -167.370 deg,	P =    -0.011 deg,	R =   -81.388 deg
};
P[1764]{
   GP1:
	UF : 7, UT : 3,	CONFIG : 'F U T, 0, 0, 0',
	X =  -311.718  mm,	Y =   108.335  mm,	Z =     0.000  mm,
	W =  -167.371 deg,	P =     0.856 deg,	R =   -94.595 deg
};
P[1765]{
   GP1:
	UF : 7, UT : 3,	CONFIG : 'F U T, 0, 0, 0',
	X =  -311.718  mm,	Y =   108.335  mm,	Z =     0.000  mm,
	W =  -167.371 deg,	P =     0.856 deg,	R =   -94.595 deg
};
P[1766]{
   GP1:
	UF : 7, UT : 3,	CONFIG : 'F U T, 0, 0, 0',
	X =  -311.718  mm,	Y =   108.335  mm,	Z =     0.000  mm,
	W =  -167.371 deg,	P =     0.856 deg,	R =   -94.595 deg
};
P[1767]{
   GP1:
	UF : 7, UT : 3,	CONFIG : 'F U T, 0, 0, 0',
	X =  -311.718  mm,	Y =   108.335  mm,	Z =     0.000  mm,
	W =  -167.371 deg,	P =     0.856 deg,	R =   -94.595 deg
};
P[1768]{
   GP1:
	UF : 7, UT : 3,	CONFIG : 'F U T, 0, 0, 0',
	X =  -308.421  mm,	Y =   117.363  mm,	Z =     0.229  mm,
	W =  -167.587 deg,	P =     1.914 deg,	R =   -95.845 deg
};
P[1769]{
   GP1:
	UF : 7, UT : 3,	CONFIG : 'F U T, 0, 0, 0',
	X =  -305.761  mm,	Y =   124.137  mm,	Z =     0.466  mm,
	W =  -167.927 deg,	P =     1.952 deg,	R =   -97.041 deg
};
P[1770]{
   GP1:
	UF : 7, UT : 3,	CONFIG : 'F U T, 0, 0, 0',
	X =  -299.660  mm,	Y =   138.219  mm,	Z =     0.736  mm,
	W =  -168.402 deg,	P =     0.599 deg,	R =   -99.739 deg
};
P[1771]{
   GP1:
	UF : 7, UT : 3,	CONFIG : 'F U T, 0, 0, 0',
	X =  -290.869  mm,	Y =   155.886  mm,	Z =     0.599  mm,
